LIN {X 0,Y 298.384,Z 335.943,A -85,B 0,C 180,E1 -16518.911,E2 -16518.911} C_VEL
LIN {X 0,Y 298.442,Z 335.935,A -85,B 0,C 180,E1 -16523.191,E2 -16523.191} C_VEL
LIN {X 0,Y 298.393,Z 335.94,A -85,B 0,C 180,E1 -16527.199,E2 -16527.199} C_VEL
LIN {X 0,Y 298.428,Z 335.937,A -85,B 0,C 180,E1 -16530.613,E2 -16530.613} C_VEL
LIN {X 0,Y 298.478,Z 335.928,A -85,B 0,C 180,E1 -16533.473,E2 -16533.473} C_VEL
LIN {X 0,Y 298.429,Z 335.938,A -85,B 0,C 180,E1 -16536.696,E2 -16536.696} C_VEL
LIN {X 0,Y 298.533,Z 335.925,A -85,B 0,C 180,E1 -16540.756,E2 -16540.756} C_VEL
LIN {X 0,Y 298.586,Z 335.915,A -85,B 0,C 180,E1 -16544.994,E2 -16544.994} C_VEL
LIN {X 0,Y 298.586,Z 335.915,A -85,B 0,C 180,E1 -16549.146,E2 -16549.146} C_VEL
LIN {X 0,Y 298.753,Z 335.894,A -85,B 0,C 180,E1 -16551.885,E2 -16551.885} C_VEL
LIN {X 0,Y 298.654,Z 335.909,A -85,B 0,C 180,E1 -16554.598,E2 -16554.598} C_VEL
LIN {X 0,Y 298.916,Z 335.876,A -85,B 0,C 180,E1 -16558.652,E2 -16558.652} C_VEL
LIN {X 0,Y 298.918,Z 335.872,A -85,B 0,C 180,E1 -16561.347,E2 -16561.347} C_VEL
LIN {X 0,Y 298.785,Z 335.89,A -85,B 0,C 180,E1 -16562.896,E2 -16562.896} C_VEL
LIN {X 0,Y 297.957,Z 335.996,A -85,B 0,C 180,E1 -16564.02,E2 -16564.02} C_VEL
LIN {X 0,Y 295.074,Z 336.353,A -85,B 0,C 180,E1 -16565.854,E2 -16565.854} C_VEL
LIN {X 0,Y 292.741,Z 336.645,A -85,B 0,C 180,E1 -16567.341,E2 -16567.341} C_VEL
LIN {X 0,Y 291.768,Z 336.766,A -85,B 0,C 180,E1 -16568.492,E2 -16568.492} C_VEL
LIN {X 0,Y 291.696,Z 336.772,A -85,B 0,C 180,E1 -16568.881,E2 -16568.881} C_VEL
LIN {X 0,Y 291.515,Z 336.798,A -85,B 0,C 180,E1 -16573.95,E2 -16573.95} C_VEL
LIN {X 0,Y 291.48,Z 336.799,A -85,B 0,C 180,E1 -16576.818,E2 -16576.818} C_VEL
LIN {X 0,Y 291.443,Z 336.806,A -85,B 0,C 180,E1 -16579.875,E2 -16579.875} C_VEL
LIN {X 0,Y 291.393,Z 336.813,A -85,B 0,C 180,E1 -16584.206,E2 -16584.206} C_VEL
LIN {X 0,Y 291.415,Z 336.807,A -85,B 0,C 180,E1 -16587.272,E2 -16587.272} C_VEL
LIN {X 0,Y 291.332,Z 336.819,A -85,B 0,C 180,E1 -16590.437,E2 -16590.437} C_VEL
LIN {X 0,Y 291.339,Z 336.821,A -85,B 0,C 180,E1 -16593.699,E2 -16593.699} C_VEL
LIN {X 0,Y 291.431,Z 336.915,A -85,B 0,C 180,E1 -16596.753,E2 -16596.753} C_VEL
LIN {X 0,Y 292.734,Z 343.937,A -85,B 0,C 180,E1 -16600.407,E2 -16600.407} C_VEL
LIN {X 0,Y 294.252,Z 351.677,A -85,B 0,C 180,E1 -16604.234,E2 -16604.234} C_VEL
LIN {X 0,Y 296.055,Z 360.385,A -85,B 0,C 180,E1 -16608.344,E2 -16608.344} C_VEL
LIN {X 0,Y 296.139,Z 362.771,A -85,B 0,C 180,E1 -16609.413,E2 -16609.413} C_VEL
LIN {X 0,Y 294.612,Z 372.008,A -85,B 0,C 180,E1 -16613.391,E2 -16613.391} C_VEL
LIN {X 0,Y 293.002,Z 383.21,A -85,B 0,C 180,E1 -16618.152,E2 -16618.152} C_VEL
LIN {X 0,Y 291.754,Z 394.182,A -85,B 0,C 180,E1 -16622.764,E2 -16622.764} C_VEL
LIN {X 0,Y 291.663,Z 395.459,A -85,B 0,C 180,E1 -16623.189,E2 -16623.189} C_VEL
LIN {X 0,Y 293.313,Z 416.036,A -85,B 0,C 180,E1 -16624.452,E2 -16624.452} C_VEL
LIN {X 0,Y 294.42,Z 430.699,A -85,B 0,C 180,E1 -16625.619,E2 -16625.619} C_VEL
LIN {X 0,Y 295.568,Z 445.292,A -85,B 0,C 180,E1 -16627.087,E2 -16627.087} C_VEL
LIN {X 0,Y 296.15,Z 455.041,A -85,B 0,C 180,E1 -16628.237,E2 -16628.237} C_VEL
LIN {X 0,Y 294.693,Z 467.515,A -85,B 0,C 180,E1 -16629.953,E2 -16629.953} C_VEL
LIN {X 0,Y 293.284,Z 478.836,A -85,B 0,C 180,E1 -16631.851,E2 -16631.851} C_VEL
LIN {X 0,Y 292.138,Z 489.112,A -85,B 0,C 180,E1 -16633.941,E2 -16633.941} C_VEL
LIN {X 0,Y 291.317,Z 497.647,A -85,B 0,C 180,E1 -16636.041,E2 -16636.041} C_VEL
LIN {X 0,Y 290.887,Z 505.868,A -85,B 0,C 180,E1 -16638.504,E2 -16638.504} C_VEL
LIN {X 0,Y 290.817,Z 512.39,A -85,B 0,C 180,E1 -16640.964,E2 -16640.964} C_VEL
LIN {X 0,Y 291.047,Z 516.816,A -85,B 0,C 180,E1 -16643.067,E2 -16643.067} C_VEL
LIN {X 0,Y 291.187,Z 519.192,A -85,B 0,C 180,E1 -16644.461,E2 -16644.461} C_VEL
LIN {X 0,Y 291.509,Z 522.595,A -85,B 0,C 180,E1 -16647.238,E2 -16647.238} C_VEL
LIN {X 0,Y 291.68,Z 523.685,A -85,B 0,C 180,E1 -16648.621,E2 -16648.621} C_VEL
LIN {X 0,Y 291.849,Z 524.383,A -85,B 0,C 180,E1 -16650.001,E2 -16650.001} C_VEL
LIN {X 0,Y 291.523,Z 524.606,A -85,B 0,C 180,E1 -16651.383,E2 -16651.383} C_VEL
LIN {X 0,Y 290.918,Z 523.938,A -85,B 0,C 180,E1 -16654.157,E2 -16654.157} C_VEL
LIN {X 0,Y 290.727,Z 523.064,A -85,B 0,C 180,E1 -16655.55,E2 -16655.55} C_VEL
LIN {X 0,Y 290.281,Z 520.217,A -85,B 0,C 180,E1 -16658.354,E2 -16658.354} C_VEL
LIN {X 0,Y 290.24,Z 515.983,A -85,B 0,C 180,E1 -16661.171,E2 -16661.171} C_VEL
LIN {X 0,Y 290.843,Z 510.353,A -85,B 0,C 180,E1 -16663.985,E2 -16663.985} C_VEL
LIN {X 0,Y 292.262,Z 503.283,A -85,B 0,C 180,E1 -16666.773,E2 -16666.773} C_VEL
LIN {X 0,Y 294.433,Z 494.668,A -85,B 0,C 180,E1 -16669.523,E2 -16669.523} C_VEL
LIN {X 0,Y 297.551,Z 484.315,A -85,B 0,C 180,E1 -16672.206,E2 -16672.206} C_VEL
LIN {X 0,Y 300.623,Z 474.827,A -85,B 0,C 180,E1 -16674.253,E2 -16674.253} C_VEL
LIN {X 0,Y 303.764,Z 464.971,A -85,B 0,C 180,E1 -16676.079,E2 -16676.079} C_VEL
LIN {X 0,Y 307.037,Z 451.397,A -85,B 0,C 180,E1 -16678.358,E2 -16678.358} C_VEL
LIN {X 0,Y 309.072,Z 440.707,A -85,B 0,C 180,E1 -16680.018,E2 -16680.018} C_VEL
LIN {X 0,Y 310.207,Z 429.791,A -85,B 0,C 180,E1 -16681.737,E2 -16681.737} C_VEL
LIN {X 0,Y 310.622,Z 419.575,A -85,B 0,C 180,E1 -16683.437,E2 -16683.437} C_VEL
LIN {X 0,Y 310.565,Z 410.326,A -85,B 0,C 180,E1 -16685.096,E2 -16685.096} C_VEL
LIN {X 0,Y 310.075,Z 400.116,A -85,B 0,C 180,E1 -16687.159,E2 -16687.159} C_VEL
LIN {X 0,Y 309.74,Z 393.575,A -85,B 0,C 180,E1 -16688.649,E2 -16688.649} C_VEL
LIN {X 0,Y 309.457,Z 385.456,A -85,B 0,C 180,E1 -16690.737,E2 -16690.737} C_VEL
LIN {X 0,Y 309.469,Z 380.582,A -85,B 0,C 180,E1 -16692.221,E2 -16692.221} C_VEL
LIN {X 0,Y 309.456,Z 378.608,A -85,B 0,C 180,E1 -16692.948,E2 -16692.948} C_VEL
LIN {X 0,Y 309.152,Z 375.079,A -85,B 0,C 180,E1 -16695.193,E2 -16695.193} C_VEL
LIN {X 0,Y 309.337,Z 373.381,A -85,B 0,C 180,E1 -16697.032,E2 -16697.032} C_VEL
LIN {X 0,Y 310.764,Z 372.281,A -85,B 0,C 180,E1 -16700.258,E2 -16700.258} C_VEL
LIN {X 0,Y 312.772,Z 372.924,A -85,B 0,C 180,E1 -16702.65,E2 -16702.65} C_VEL
LIN {X 0,Y 314.831,Z 374.395,A -85,B 0,C 180,E1 -16704.522,E2 -16704.522} C_VEL
LIN {X 0,Y 317.095,Z 376.765,A -85,B 0,C 180,E1 -16706.352,E2 -16706.352} C_VEL
LIN {X 0,Y 318.444,Z 379.308,A -85,B 0,C 180,E1 -16707.599,E2 -16707.599} C_VEL
LIN {X 0,Y 319.816,Z 385.394,A -85,B 0,C 180,E1 -16709.641,E2 -16709.641} C_VEL
LIN {X 0,Y 320.499,Z 391.158,A -85,B 0,C 180,E1 -16711.3,E2 -16711.3} C_VEL
LIN {X 0,Y 316.891,Z 401.154,A -85,B 0,C 180,E1 -16712.958,E2 -16712.958} C_VEL
LIN {X 0,Y 312.724,Z 411.585,A -85,B 0,C 180,E1 -16715.079,E2 -16715.079} C_VEL
LIN {X 0,Y 308.879,Z 420.286,A -85,B 0,C 180,E1 -16717.244,E2 -16717.244} C_VEL
LIN {X 0,Y 305.859,Z 426.538,A -85,B 0,C 180,E1 -16719.136,E2 -16719.136} C_VEL
LIN {X 0,Y 302.504,Z 433.284,A -85,B 0,C 180,E1 -16721.721,E2 -16721.721} C_VEL
LIN {X 0,Y 299.864,Z 438.042,A -85,B 0,C 180,E1 -16724.09,E2 -16724.09} C_VEL
LIN {X 0,Y 297.743,Z 441.439,A -85,B 0,C 180,E1 -16726.347,E2 -16726.347} C_VEL
LIN {X 0,Y 295.668,Z 444.227,A -85,B 0,C 180,E1 -16729.038,E2 -16729.038} C_VEL
LIN {X 0,Y 294.017,Z 445.702,A -85,B 0,C 180,E1 -16731.755,E2 -16731.755} C_VEL
LIN {X 0,Y 292.837,Z 445.876,A -85,B 0,C 180,E1 -16734.492,E2 -16734.492} C_VEL
LIN {X 0,Y 292.076,Z 444.754,A -85,B 0,C 180,E1 -16737.242,E2 -16737.242} C_VEL
LIN {X 0,Y 291.759,Z 442.304,A -85,B 0,C 180,E1 -16740,E2 -16740} C_VEL
LIN {X 0,Y 291.643,Z 439.625,A -85,B 0,C 180,E1 -16742.072,E2 -16742.072} C_VEL
LIN {X 0,Y 291.566,Z 434.76,A -85,B 0,C 180,E1 -16744.84,E2 -16744.84} C_VEL
LIN {X 0,Y 292.038,Z 430.099,A -85,B 0,C 180,E1 -16746.911,E2 -16746.911} C_VEL
LIN {X 0,Y 292.606,Z 423.431,A -85,B 0,C 180,E1 -16749.331,E2 -16749.331} C_VEL
LIN {X 0,Y 293.372,Z 415.255,A -85,B 0,C 180,E1 -16751.749,E2 -16751.749} C_VEL
LIN {X 0,Y 294.492,Z 405.302,A -85,B 0,C 180,E1 -16754.159,E2 -16754.159} C_VEL
LIN {X 0,Y 295.596,Z 395.056,A -85,B 0,C 180,E1 -16756.223,E2 -16756.223} C_VEL
LIN {X 0,Y 297.097,Z 382.921,A -85,B 0,C 180,E1 -16758.244,E2 -16758.244} C_VEL
LIN {X 0,Y 298.434,Z 370.378,A -85,B 0,C 180,E1 -16759.967,E2 -16759.967} C_VEL
LIN {X 0,Y 298.882,Z 363.575,A -85,B 0,C 180,E1 -16760.784,E2 -16760.784} C_VEL
LIN {X 0,Y 295.194,Z 350.343,A -85,B 0,C 180,E1 -16762.392,E2 -16762.392} C_VEL
LIN {X 0,Y 291.55,Z 337.403,A -85,B 0,C 180,E1 -16763.773,E2 -16763.773} C_VEL
LIN {X 0,Y 291.45,Z 336.845,A -85,B 0,C 180,E1 -16764.017,E2 -16764.017} C_VEL
LIN {X 0,Y 291.431,Z 336.807,A -85,B 0,C 180,E1 -16767.271,E2 -16767.271} C_VEL
LIN {X 0,Y 291.343,Z 336.82,A -85,B 0,C 180,E1 -16770.437,E2 -16770.437} C_VEL
LIN {X 0,Y 291.35,Z 336.816,A -85,B 0,C 180,E1 -16773.698,E2 -16773.698} C_VEL
LIN {X 0,Y 291.381,Z 336.811,A -85,B 0,C 180,E1 -16777.254,E2 -16777.254} C_VEL
LIN {X 0,Y 291.338,Z 336.821,A -85,B 0,C 180,E1 -16780.642,E2 -16780.642} C_VEL
LIN {X 0,Y 291.296,Z 336.826,A -85,B 0,C 180,E1 -16784.402,E2 -16784.402} C_VEL
LIN {X 0,Y 291.361,Z 336.819,A -85,B 0,C 180,E1 -16788.397,E2 -16788.397} C_VEL
LIN {X 0,Y 291.38,Z 336.812,A -85,B 0,C 180,E1 -16791.161,E2 -16791.161} C_VEL
LIN {X 0,Y 291.392,Z 336.812,A -85,B 0,C 180,E1 -16794.629,E2 -16794.629} C_VEL
LIN {X 0,Y 291.377,Z 336.815,A -85,B 0,C 180,E1 -16797.95,E2 -16797.95} C_VEL
LIN {X 0,Y 291.383,Z 336.811,A -85,B 0,C 180,E1 -16801.157,E2 -16801.157} C_VEL
LIN {X 0,Y 291.42,Z 336.811,A -85,B 0,C 180,E1 -16804.271,E2 -16804.271} C_VEL
LIN {X 0,Y 291.38,Z 336.812,A -85,B 0,C 180,E1 -16807.298,E2 -16807.298} C_VEL
LIN {X 0,Y 291.463,Z 336.803,A -85,B 0,C 180,E1 -16810.269,E2 -16810.269} C_VEL
LIN {X 0,Y 291.561,Z 336.79,A -85,B 0,C 180,E1 -16814.623,E2 -16814.623} C_VEL
LIN {X 0,Y 291.542,Z 336.79,A -85,B 0,C 180,E1 -16818.88,E2 -16818.88} C_VEL
LIN {X 0,Y 291.714,Z 336.773,A -85,B 0,C 180,E1 -16821.687,E2 -16821.687} C_VEL
LIN {X 0,Y 291.635,Z 336.78,A -85,B 0,C 180,E1 -16824.467,E2 -16824.467} C_VEL
LIN {X 0,Y 291.893,Z 336.747,A -85,B 0,C 180,E1 -16828.619,E2 -16828.619} C_VEL
LIN {X 0,Y 291.893,Z 336.75,A -85,B 0,C 180,E1 -16831.378,E2 -16831.378} C_VEL
LIN {X 0,Y 291.75,Z 336.765,A -85,B 0,C 180,E1 -16836.916,E2 -16836.916} C_VEL
LIN {X 0,Y 291.632,Z 336.784,A -85,B 0,C 180,E1 -16839.71,E2 -16839.71} C_VEL
LIN {X 0,Y 291.525,Z 336.794,A -85,B 0,C 180,E1 -16843.949,E2 -16843.949} C_VEL
LIN {X 0,Y 291.489,Z 336.798,A -85,B 0,C 180,E1 -16846.816,E2 -16846.816} C_VEL
LIN {X 0,Y 291.452,Z 336.804,A -85,B 0,C 180,E1 -16849.873,E2 -16849.873} C_VEL
LIN {X 0,Y 291.4,Z 336.809,A -85,B 0,C 180,E1 -16854.204,E2 -16854.204} C_VEL
LIN {X 0,Y 291.419,Z 336.811,A -85,B 0,C 180,E1 -16857.27,E2 -16857.27} C_VEL
LIN {X 0,Y 291.334,Z 336.817,A -85,B 0,C 180,E1 -16860.436,E2 -16860.436} C_VEL
LIN {X 0,Y 291.343,Z 336.818,A -85,B 0,C 180,E1 -16863.697,E2 -16863.697} C_VEL
LIN {X 0,Y 291.371,Z 336.817,A -85,B 0,C 180,E1 -16867.252,E2 -16867.252} C_VEL
LIN {X 0,Y 291.33,Z 336.818,A -85,B 0,C 180,E1 -16870.641,E2 -16870.641} C_VEL
LIN {X 0,Y 291.31,Z 336.821,A -85,B 0,C 180,E1 -16874.396,E2 -16874.396} C_VEL
LIN {X 0,Y 291.323,Z 336.819,A -85,B 0,C 180,E1 -16878.403,E2 -16878.403} C_VEL
LIN {X 0,Y 291.349,Z 336.819,A -85,B 0,C 180,E1 -16881.157,E2 -16881.157} C_VEL
LIN {X 0,Y 291.356,Z 336.817,A -85,B 0,C 180,E1 -16884.625,E2 -16884.625} C_VEL
LIN {X 0,Y 291.37,Z 336.812,A -85,B 0,C 180,E1 -16887.95,E2 -16887.95} C_VEL
LIN {X 0,Y 291.378,Z 336.814,A -85,B 0,C 180,E1 -16891.157,E2 -16891.157} C_VEL
LIN {X 0,Y 291.411,Z 336.809,A -85,B 0,C 180,E1 -16894.271,E2 -16894.271} C_VEL
LIN {X 0,Y 291.376,Z 336.813,A -85,B 0,C 180,E1 -16897.299,E2 -16897.299} C_VEL
LIN {X 0,Y 291.451,Z 336.805,A -85,B 0,C 180,E1 -16900.269,E2 -16900.269} C_VEL
LIN {X 0,Y 291.548,Z 336.795,A -85,B 0,C 180,E1 -16904.623,E2 -16904.623} C_VEL
LIN {X 0,Y 291.53,Z 336.795,A -85,B 0,C 180,E1 -16908.88,E2 -16908.88} C_VEL
LIN {X 0,Y 291.703,Z 336.771,A -85,B 0,C 180,E1 -16911.688,E2 -16911.688} C_VEL
LIN {X 0,Y 291.625,Z 336.785,A -85,B 0,C 180,E1 -16914.468,E2 -16914.468} C_VEL
LIN {X 0,Y 291.883,Z 336.752,A -85,B 0,C 180,E1 -16918.62,E2 -16918.62} C_VEL
LIN {X 0,Y 291.884,Z 336.748,A -85,B 0,C 180,E1 -16921.379,E2 -16921.379} C_VEL
LIN {X 0,Y 291.739,Z 336.768,A -85,B 0,C 180,E1 -16926.918,E2 -16926.918} C_VEL
LIN {X 0,Y 291.696,Z 336.772,A -85,B 0,C 180,E1 -16928.881,E2 -16928.881} C_VEL
LIN {X 0,Y 291.026,Z 336.859,A -85,B 0,C 180,E1 -16930.033,E2 -16930.033} C_VEL
LIN {X 0,Y 288.091,Z 337.223,A -85,B 0,C 180,E1 -16931.906,E2 -16931.906} C_VEL
LIN {X 0,Y 285.6,Z 337.534,A -85,B 0,C 180,E1 -16933.427,E2 -16933.427} C_VEL
LIN {X 0,Y 284.543,Z 337.666,A -85,B 0,C 180,E1 -16934.608,E2 -16934.608} C_VEL
LIN {X 0,Y 284.464,Z 337.673,A -85,B 0,C 180,E1 -16935.008,E2 -16935.008} C_VEL
LIN {X 0,Y 284.396,Z 337.681,A -85,B 0,C 180,E1 -16938.739,E2 -16938.739} C_VEL
LIN {X 0,Y 284.359,Z 337.687,A -85,B 0,C 180,E1 -16943.293,E2 -16943.293} C_VEL
LIN {X 0,Y 284.39,Z 337.682,A -85,B 0,C 180,E1 -16947.174,E2 -16947.174} C_VEL
LIN {X 0,Y 284.291,Z 337.695,A -85,B 0,C 180,E1 -16951.275,E2 -16951.275} C_VEL
LIN {X 0,Y 284.356,Z 337.69,A -85,B 0,C 180,E1 -16955.355,E2 -16955.355} C_VEL
LIN {X 0,Y 284.414,Z 337.85,A -85,B 0,C 180,E1 -16956.484,E2 -16956.484} C_VEL
LIN {X 0,Y 285.934,Z 346.081,A -85,B 0,C 180,E1 -16960.841,E2 -16960.841} C_VEL
LIN {X 0,Y 287.642,Z 354.606,A -85,B 0,C 180,E1 -16965.118,E2 -16965.118} C_VEL
LIN {X 0,Y 289.075,Z 361.67,A -85,B 0,C 180,E1 -16968.512,E2 -16968.512} C_VEL
LIN {X 0,Y 288.92,Z 364.669,A -85,B 0,C 180,E1 -16969.865,E2 -16969.865} C_VEL
LIN {X 0,Y 287.32,Z 373.641,A -85,B 0,C 180,E1 -16973.823,E2 -16973.823} C_VEL
LIN {X 0,Y 285.916,Z 383.442,A -85,B 0,C 180,E1 -16978.099,E2 -16978.099} C_VEL
LIN {X 0,Y 284.641,Z 394.497,A -85,B 0,C 180,E1 -16982.794,E2 -16982.794} C_VEL
LIN {X 0,Y 285.142,Z 401.706,A -85,B 0,C 180,E1 -16983.236,E2 -16983.236} C_VEL
LIN {X 0,Y 286.343,Z 416.546,A -85,B 0,C 180,E1 -16984.208,E2 -16984.208} C_VEL
LIN {X 0,Y 287.461,Z 432.159,A -85,B 0,C 180,E1 -16985.539,E2 -16985.539} C_VEL
LIN {X 0,Y 288.566,Z 446.524,A -85,B 0,C 180,E1 -16987.067,E2 -16987.067} C_VEL
LIN {X 0,Y 288.999,Z 456.415,A -85,B 0,C 180,E1 -16988.308,E2 -16988.308} C_VEL
LIN {X 0,Y 287.363,Z 469.079,A -85,B 0,C 180,E1 -16990.165,E2 -16990.165} C_VEL
LIN {X 0,Y 286.009,Z 479.977,A -85,B 0,C 180,E1 -16992.113,E2 -16992.113} C_VEL
LIN {X 0,Y 284.908,Z 489.858,A -85,B 0,C 180,E1 -16994.257,E2 -16994.257} C_VEL
LIN {X 0,Y 284.185,Z 498.091,A -85,B 0,C 180,E1 -16996.413,E2 -16996.413} C_VEL
LIN {X 0,Y 283.861,Z 504.96,A -85,B 0,C 180,E1 -16998.577,E2 -16998.577} C_VEL
LIN {X 0,Y 283.818,Z 510.593,A -85,B 0,C 180,E1 -17000.739,E2 -17000.739} C_VEL
LIN {X 0,Y 284.019,Z 515.128,A -85,B 0,C 180,E1 -17002.894,E2 -17002.894} C_VEL
LIN {X 0,Y 284.245,Z 518.631,A -85,B 0,C 180,E1 -17005.037,E2 -17005.037} C_VEL
LIN {X 0,Y 284.512,Z 521.176,A -85,B 0,C 180,E1 -17007.17,E2 -17007.17} C_VEL
LIN {X 0,Y 284.695,Z 522.34,A -85,B 0,C 180,E1 -17008.587,E2 -17008.587} C_VEL
LIN {X 0,Y 284.862,Z 523.099,A -85,B 0,C 180,E1 -17010.001,E2 -17010.001} C_VEL
LIN {X 0,Y 284.501,Z 523.377,A -85,B 0,C 180,E1 -17011.417,E2 -17011.417} C_VEL
LIN {X 0,Y 283.867,Z 522.826,A -85,B 0,C 180,E1 -17014.261,E2 -17014.261} C_VEL
LIN {X 0,Y 283.664,Z 522.015,A -85,B 0,C 180,E1 -17015.689,E2 -17015.689} C_VEL
LIN {X 0,Y 283.179,Z 519.302,A -85,B 0,C 180,E1 -17018.565,E2 -17018.565} C_VEL
LIN {X 0,Y 283.18,Z 515.227,A -85,B 0,C 180,E1 -17021.453,E2 -17021.453} C_VEL
LIN {X 0,Y 283.878,Z 509.787,A -85,B 0,C 180,E1 -17024.335,E2 -17024.335} C_VEL
LIN {X 0,Y 285.411,Z 502.934,A -85,B 0,C 180,E1 -17027.188,E2 -17027.188} C_VEL
LIN {X 0,Y 287.698,Z 494.586,A -85,B 0,C 180,E1 -17030,E2 -17030} C_VEL
LIN {X 0,Y 290.995,Z 484.598,A -85,B 0,C 180,E1 -17032.733,E2 -17032.733} C_VEL
LIN {X 0,Y 294.157,Z 475.6,A -85,B 0,C 180,E1 -17034.784,E2 -17034.784} C_VEL
LIN {X 0,Y 297.475,Z 466.005,A -85,B 0,C 180,E1 -17036.673,E2 -17036.673} C_VEL
LIN {X 0,Y 301.507,Z 451.11,A -85,B 0,C 180,E1 -17039.309,E2 -17039.309} C_VEL
LIN {X 0,Y 303.718,Z 440.158,A -85,B 0,C 180,E1 -17041.11,E2 -17041.11} C_VEL
LIN {X 0,Y 305.168,Z 427.686,A -85,B 0,C 180,E1 -17043.237,E2 -17043.237} C_VEL
LIN {X 0,Y 305.763,Z 415.971,A -85,B 0,C 180,E1 -17045.396,E2 -17045.396} C_VEL
LIN {X 0,Y 305.801,Z 406.067,A -85,B 0,C 180,E1 -17047.462,E2 -17047.462} C_VEL
LIN {X 0,Y 305.758,Z 398.289,A -85,B 0,C 180,E1 -17049.308,E2 -17049.308} C_VEL
LIN {X 0,Y 305.929,Z 390.966,A -85,B 0,C 180,E1 -17051.249,E2 -17051.249} C_VEL
LIN {X 0,Y 306.187,Z 386.252,A -85,B 0,C 180,E1 -17052.735,E2 -17052.735} C_VEL
LIN {X 0,Y 306.259,Z 384.286,A -85,B 0,C 180,E1 -17053.508,E2 -17053.508} C_VEL
LIN {X 0,Y 306.166,Z 381.437,A -85,B 0,C 180,E1 -17055.367,E2 -17055.367} C_VEL
LIN {X 0,Y 306.376,Z 379.73,A -85,B 0,C 180,E1 -17057.228,E2 -17057.228} C_VEL
LIN {X 0,Y 307.597,Z 378.679,A -85,B 0,C 180,E1 -17060.227,E2 -17060.227} C_VEL
LIN {X 0,Y 309.46,Z 379.193,A -85,B 0,C 180,E1 -17062.644,E2 -17062.644} C_VEL
LIN {X 0,Y 311.184,Z 380.466,A -85,B 0,C 180,E1 -17064.396,E2 -17064.396} C_VEL
LIN {X 0,Y 313.1,Z 382.536,A -85,B 0,C 180,E1 -17066.154,E2 -17066.154} C_VEL
LIN {X 0,Y 313.799,Z 383.681,A -85,B 0,C 180,E1 -17066.841,E2 -17066.841} C_VEL
LIN {X 0,Y 314.759,Z 388.181,A -85,B 0,C 180,E1 -17068.564,E2 -17068.564} C_VEL
LIN {X 0,Y 315.385,Z 393.682,A -85,B 0,C 180,E1 -17070.352,E2 -17070.352} C_VEL
LIN {X 0,Y 315.358,Z 394.716,A -85,B 0,C 180,E1 -17070.641,E2 -17070.641} C_VEL
LIN {X 0,Y 311.502,Z 404.333,A -85,B 0,C 180,E1 -17072.318,E2 -17072.318} C_VEL
LIN {X 0,Y 306.887,Z 414.87,A -85,B 0,C 180,E1 -17074.571,E2 -17074.571} C_VEL
LIN {X 0,Y 302.852,Z 423.182,A -85,B 0,C 180,E1 -17076.765,E2 -17076.765} C_VEL
LIN {X 0,Y 299.687,Z 429.143,A -85,B 0,C 180,E1 -17078.685,E2 -17078.685} C_VEL
LIN {X 0,Y 296.129,Z 435.545,A -85,B 0,C 180,E1 -17081.314,E2 -17081.314} C_VEL
LIN {X 0,Y 293.115,Z 440.386,A -85,B 0,C 180,E1 -17083.945,E2 -17083.945} C_VEL
LIN {X 0,Y 291.096,Z 443.279,A -85,B 0,C 180,E1 -17086.029,E2 -17086.029} C_VEL
LIN {X 0,Y 288.881,Z 445.824,A -85,B 0,C 180,E1 -17088.777,E2 -17088.777} C_VEL
LIN {X 0,Y 287.127,Z 447.093,A -85,B 0,C 180,E1 -17091.555,E2 -17091.555} C_VEL
LIN {X 0,Y 285.87,Z 447.083,A -85,B 0,C 180,E1 -17094.357,E2 -17094.357} C_VEL
LIN {X 0,Y 285.062,Z 445.784,A -85,B 0,C 180,E1 -17097.174,E2 -17097.174} C_VEL
LIN {X 0,Y 284.735,Z 443.163,A -85,B 0,C 180,E1 -17100,E2 -17100} C_VEL
LIN {X 0,Y 284.581,Z 440.331,A -85,B 0,C 180,E1 -17102.123,E2 -17102.123} C_VEL
LIN {X 0,Y 284.355,Z 436.732,A -85,B 0,C 180,E1 -17104.253,E2 -17104.253} C_VEL
LIN {X 0,Y 285.018,Z 430.476,A -85,B 0,C 180,E1 -17107.082,E2 -17107.082} C_VEL
LIN {X 0,Y 285.686,Z 422.524,A -85,B 0,C 180,E1 -17109.916,E2 -17109.916} C_VEL
LIN {X 0,Y 286.56,Z 413.933,A -85,B 0,C 180,E1 -17112.392,E2 -17112.392} C_VEL
LIN {X 0,Y 287.566,Z 405.099,A -85,B 0,C 180,E1 -17114.508,E2 -17114.508} C_VEL
LIN {X 0,Y 288.736,Z 394.623,A -85,B 0,C 180,E1 -17116.619,E2 -17116.619} C_VEL
LIN {X 0,Y 290.253,Z 382.41,A -85,B 0,C 180,E1 -17118.644,E2 -17118.644} C_VEL
LIN {X 0,Y 291.665,Z 369.239,A -85,B 0,C 180,E1 -17120.451,E2 -17120.451} C_VEL
LIN {X 0,Y 291.914,Z 364.846,A -85,B 0,C 180,E1 -17120.986,E2 -17120.986} C_VEL
LIN {X 0,Y 288.439,Z 352.306,A -85,B 0,C 180,E1 -17122.56,E2 -17122.56} C_VEL
LIN {X 0,Y 284.538,Z 338.361,A -85,B 0,C 180,E1 -17124.085,E2 -17124.085} C_VEL
LIN {X 0,Y 284.401,Z 337.718,A -85,B 0,C 180,E1 -17124.367,E2 -17124.367} C_VEL
LIN {X 0,Y 284.34,Z 337.691,A -85,B 0,C 180,E1 -17128.01,E2 -17128.01} C_VEL
LIN {X 0,Y 284.301,Z 337.695,A -85,B 0,C 180,E1 -17131.274,E2 -17131.274} C_VEL
LIN {X 0,Y 284.346,Z 337.688,A -85,B 0,C 180,E1 -17135.348,E2 -17135.348} C_VEL
LIN {X 0,Y 284.318,Z 337.693,A -85,B 0,C 180,E1 -17138.169,E2 -17138.169} C_VEL
LIN {X 0,Y 284.275,Z 337.699,A -85,B 0,C 180,E1 -17142.124,E2 -17142.124} C_VEL
LIN {X 0,Y 284.278,Z 337.698,A -85,B 0,C 180,E1 -17146.192,E2 -17146.192} C_VEL
LIN {X 0,Y 284.357,Z 337.689,A -85,B 0,C 180,E1 -17150.013,E2 -17150.013} C_VEL
LIN {X 0,Y 284.36,Z 337.686,A -85,B 0,C 180,E1 -17153.617,E2 -17153.617} C_VEL
LIN {X 0,Y 284.313,Z 337.692,A -85,B 0,C 180,E1 -17157.189,E2 -17157.189} C_VEL
LIN {X 0,Y 284.361,Z 337.689,A -85,B 0,C 180,E1 -17160.375,E2 -17160.375} C_VEL
LIN {X 0,Y 284.381,Z 337.684,A -85,B 0,C 180,E1 -17163.586,E2 -17163.586} C_VEL
LIN {X 0,Y 284.339,Z 337.69,A -85,B 0,C 180,E1 -17166.703,E2 -17166.703} C_VEL
LIN {X 0,Y 284.409,Z 337.679,A -85,B 0,C 180,E1 -17171.261,E2 -17171.261} C_VEL
LIN {X 0,Y 284.498,Z 337.67,A -85,B 0,C 180,E1 -17174.458,E2 -17174.458} C_VEL
LIN {X 0,Y 284.494,Z 337.669,A -85,B 0,C 180,E1 -17178.6,E2 -17178.6} C_VEL
LIN {X 0,Y 284.665,Z 337.65,A -85,B 0,C 180,E1 -17181.48,E2 -17181.48} C_VEL
LIN {X 0,Y 284.606,Z 337.657,A -85,B 0,C 180,E1 -17184.33,E2 -17184.33} C_VEL
LIN {X 0,Y 284.859,Z 337.623,A -85,B 0,C 180,E1 -17188.585,E2 -17188.585} C_VEL
LIN {X 0,Y 284.859,Z 337.626,A -85,B 0,C 180,E1 -17191.412,E2 -17191.412} C_VEL
LIN {X 0,Y 284.702,Z 337.643,A -85,B 0,C 180,E1 -17197.089,E2 -17197.089} C_VEL
LIN {X 0,Y 284.57,Z 337.662,A -85,B 0,C 180,E1 -17199.954,E2 -17199.954} C_VEL
LIN {X 0,Y 284.484,Z 337.67,A -85,B 0,C 180,E1 -17204.301,E2 -17204.301} C_VEL
LIN {X 0,Y 284.427,Z 337.68,A -85,B 0,C 180,E1 -17207.247,E2 -17207.247} C_VEL
LIN {X 0,Y 284.38,Z 337.684,A -85,B 0,C 180,E1 -17210.241,E2 -17210.241} C_VEL
LIN {X 0,Y 284.37,Z 337.685,A -85,B 0,C 180,E1 -17213.874,E2 -17213.874} C_VEL
LIN {X 0,Y 284.394,Z 337.685,A -85,B 0,C 180,E1 -17217.171,E2 -17217.171} C_VEL
LIN {X 0,Y 284.293,Z 337.698,A -85,B 0,C 180,E1 -17221.273,E2 -17221.273} C_VEL
LIN {X 0,Y 284.339,Z 337.693,A -85,B 0,C 180,E1 -17225.346,E2 -17225.346} C_VEL
LIN {X 0,Y 284.306,Z 337.693,A -85,B 0,C 180,E1 -17228.168,E2 -17228.168} C_VEL
LIN {X 0,Y 284.267,Z 337.697,A -85,B 0,C 180,E1 -17232.123,E2 -17232.123} C_VEL
LIN {X 0,Y 284.265,Z 337.698,A -85,B 0,C 180,E1 -17236.19,E2 -17236.19} C_VEL
LIN {X 0,Y 284.302,Z 337.692,A -85,B 0,C 180,E1 -17240.022,E2 -17240.022} C_VEL
LIN {X 0,Y 284.328,Z 337.691,A -85,B 0,C 180,E1 -17243.613,E2 -17243.613} C_VEL
LIN {X 0,Y 284.304,Z 337.694,A -85,B 0,C 180,E1 -17247.188,E2 -17247.188} C_VEL
LIN {X 0,Y 284.354,Z 337.688,A -85,B 0,C 180,E1 -17250.375,E2 -17250.375} C_VEL
LIN {X 0,Y 284.372,Z 337.685,A -85,B 0,C 180,E1 -17253.586,E2 -17253.586} C_VEL
LIN {X 0,Y 284.361,Z 337.69,A -85,B 0,C 180,E1 -17256.706,E2 -17256.706} C_VEL
LIN {X 0,Y 284.397,Z 337.682,A -85,B 0,C 180,E1 -17261.261,E2 -17261.261} C_VEL
LIN {X 0,Y 284.485,Z 337.674,A -85,B 0,C 180,E1 -17264.458,E2 -17264.458} C_VEL
LIN {X 0,Y 284.481,Z 337.676,A -85,B 0,C 180,E1 -17268.601,E2 -17268.601} C_VEL
LIN {X 0,Y 284.653,Z 337.649,A -85,B 0,C 180,E1 -17271.481,E2 -17271.481} C_VEL
LIN {X 0,Y 284.595,Z 337.659,A -85,B 0,C 180,E1 -17274.331,E2 -17274.331} C_VEL
LIN {X 0,Y 284.849,Z 337.629,A -85,B 0,C 180,E1 -17278.586,E2 -17278.586} C_VEL
LIN {X 0,Y 284.85,Z 337.624,A -85,B 0,C 180,E1 -17281.413,E2 -17281.413} C_VEL
LIN {X 0,Y 284.691,Z 337.645,A -85,B 0,C 180,E1 -17287.09,E2 -17287.09} C_VEL
LIN {X 0,Y 284.559,Z 337.663,A -85,B 0,C 180,E1 -17289.955,E2 -17289.955} C_VEL
LIN {X 0,Y 284.475,Z 337.676,A -85,B 0,C 180,E1 -17294.303,E2 -17294.303} C_VEL
LIN {X 0,Y 284.464,Z 337.673,A -85,B 0,C 180,E1 -17295.008,E2 -17295.008} C_VEL
LIN {X 0,Y 283.805,Z 337.76,A -85,B 0,C 180,E1 -17296.19,E2 -17296.19} C_VEL
LIN {X 0,Y 280.909,Z 338.12,A -85,B 0,C 180,E1 -17298.112,E2 -17298.112} C_VEL
LIN {X 0,Y 278.43,Z 338.426,A -85,B 0,C 180,E1 -17299.674,E2 -17299.674} C_VEL
LIN {X 0,Y 277.354,Z 338.559,A -85,B 0,C 180,E1 -17300.885,E2 -17300.885} C_VEL
LIN {X 0,Y 277.26,Z 338.569,A -85,B 0,C 180,E1 -17301.296,E2 -17301.296} C_VEL
LIN {X 0,Y 277.312,Z 338.568,A -85,B 0,C 180,E1 -17304.171,E2 -17304.171} C_VEL
LIN {X 0,Y 277.319,Z 338.564,A -85,B 0,C 180,E1 -17307.506,E2 -17307.506} C_VEL
LIN {X 0,Y 277.265,Z 338.571,A -85,B 0,C 180,E1 -17310.482,E2 -17310.482} C_VEL
LIN {X 0,Y 277.248,Z 338.577,A -85,B 0,C 180,E1 -17313.895,E2 -17313.895} C_VEL
LIN {X 0,Y 277.35,Z 338.649,A -85,B 0,C 180,E1 -17316.12,E2 -17316.12} C_VEL
LIN {X 0,Y 278.649,Z 345.78,A -85,B 0,C 180,E1 -17320.022,E2 -17320.022} C_VEL
LIN {X 0,Y 280.385,Z 354.574,A -85,B 0,C 180,E1 -17324.574,E2 -17324.574} C_VEL
LIN {X 0,Y 281.994,Z 362.314,A -85,B 0,C 180,E1 -17328.389,E2 -17328.389} C_VEL
LIN {X 0,Y 281.917,Z 364.901,A -85,B 0,C 180,E1 -17329.599,E2 -17329.599} C_VEL
LIN {X 0,Y 280.445,Z 373.075,A -85,B 0,C 180,E1 -17333.314,E2 -17333.314} C_VEL
LIN {X 0,Y 278.834,Z 383.615,A -85,B 0,C 180,E1 -17338.043,E2 -17338.043} C_VEL
LIN {X 0,Y 277.636,Z 393.612,A -85,B 0,C 180,E1 -17342.406,E2 -17342.406} C_VEL
LIN {X 0,Y 279.204,Z 415.24,A -85,B 0,C 180,E1 -17343.836,E2 -17343.836} C_VEL
LIN {X 0,Y 280.277,Z 430.557,A -85,B 0,C 180,E1 -17345.166,E2 -17345.166} C_VEL
LIN {X 0,Y 281.344,Z 445.028,A -85,B 0,C 180,E1 -17346.736,E2 -17346.736} C_VEL
LIN {X 0,Y 282.006,Z 455.247,A -85,B 0,C 180,E1 -17348.05,E2 -17348.05} C_VEL
LIN {X 0,Y 280.476,Z 467.253,A -85,B 0,C 180,E1 -17349.848,E2 -17349.848} C_VEL
LIN {X 0,Y 279.206,Z 477.313,A -85,B 0,C 180,E1 -17351.662,E2 -17351.662} C_VEL
LIN {X 0,Y 278.064,Z 487.463,A -85,B 0,C 180,E1 -17353.859,E2 -17353.859} C_VEL
LIN {X 0,Y 277.244,Z 495.895,A -85,B 0,C 180,E1 -17356.066,E2 -17356.066} C_VEL
LIN {X 0,Y 276.853,Z 504.005,A -85,B 0,C 180,E1 -17358.655,E2 -17358.655} C_VEL
LIN {X 0,Y 276.857,Z 510.422,A -85,B 0,C 180,E1 -17361.241,E2 -17361.241} C_VEL
LIN {X 0,Y 277.09,Z 514.759,A -85,B 0,C 180,E1 -17363.448,E2 -17363.448} C_VEL
LIN {X 0,Y 277.33,Z 518.019,A -85,B 0,C 180,E1 -17365.641,E2 -17365.641} C_VEL
LIN {X 0,Y 277.516,Z 519.675,A -85,B 0,C 180,E1 -17367.098,E2 -17367.098} C_VEL
LIN {X 0,Y 277.729,Z 520.923,A -85,B 0,C 180,E1 -17368.551,E2 -17368.551} C_VEL
LIN {X 0,Y 277.893,Z 521.757,A -85,B 0,C 180,E1 -17370.001,E2 -17370.001} C_VEL
LIN {X 0,Y 277.513,Z 522.1,A -85,B 0,C 180,E1 -17371.452,E2 -17371.452} C_VEL
LIN {X 0,Y 276.818,Z 521.679,A -85,B 0,C 180,E1 -17374.369,E2 -17374.369} C_VEL
LIN {X 0,Y 276.604,Z 520.937,A -85,B 0,C 180,E1 -17375.834,E2 -17375.834} C_VEL
LIN {X 0,Y 276.099,Z 518.363,A -85,B 0,C 180,E1 -17378.786,E2 -17378.786} C_VEL
LIN {X 0,Y 276.129,Z 514.456,A -85,B 0,C 180,E1 -17381.75,E2 -17381.75} C_VEL
LIN {X 0,Y 276.916,Z 509.223,A -85,B 0,C 180,E1 -17384.703,E2 -17384.703} C_VEL
LIN {X 0,Y 278.563,Z 502.624,A -85,B 0,C 180,E1 -17387.624,E2 -17387.624} C_VEL
LIN {X 0,Y 280.996,Z 494.575,A -85,B 0,C 180,E1 -17390.498,E2 -17390.498} C_VEL
LIN {X 0,Y 284.472,Z 484.927,A -85,B 0,C 180,E1 -17393.285,E2 -17393.285} C_VEL
LIN {X 0,Y 287.703,Z 476.484,A -85,B 0,C 180,E1 -17395.334,E2 -17395.334} C_VEL
LIN {X 0,Y 291.231,Z 467.099,A -85,B 0,C 180,E1 -17397.292,E2 -17397.292} C_VEL
LIN {X 0,Y 294.985,Z 454.79,A -85,B 0,C 180,E1 -17399.629,E2 -17399.629} C_VEL
LIN {X 0,Y 297.706,Z 444.068,A -85,B 0,C 180,E1 -17401.503,E2 -17401.503} C_VEL
LIN {X 0,Y 299.414,Z 433.995,A -85,B 0,C 180,E1 -17403.316,E2 -17403.316} C_VEL
LIN {X 0,Y 300.678,Z 422.339,A -85,B 0,C 180,E1 -17405.532,E2 -17405.532} C_VEL
LIN {X 0,Y 301.252,Z 412.463,A -85,B 0,C 180,E1 -17407.646,E2 -17407.646} C_VEL
LIN {X 0,Y 301.681,Z 403.711,A -85,B 0,C 180,E1 -17409.756,E2 -17409.756} C_VEL
LIN {X 0,Y 302.265,Z 395.914,A -85,B 0,C 180,E1 -17411.924,E2 -17411.924} C_VEL
LIN {X 0,Y 302.847,Z 390.814,A -85,B 0,C 180,E1 -17413.651,E2 -17413.651} C_VEL
LIN {X 0,Y 302.902,Z 388.551,A -85,B 0,C 180,E1 -17414.921,E2 -17414.921} C_VEL
LIN {X 0,Y 302.96,Z 387.231,A -85,B 0,C 180,E1 -17415.984,E2 -17415.984} C_VEL
LIN {X 0,Y 303.242,Z 385.792,A -85,B 0,C 180,E1 -17417.873,E2 -17417.873} C_VEL
LIN {X 0,Y 303.959,Z 385.093,A -85,B 0,C 180,E1 -17419.732,E2 -17419.732} C_VEL
LIN {X 0,Y 305.135,Z 385.024,A -85,B 0,C 180,E1 -17421.547,E2 -17421.547} C_VEL
LIN {X 0,Y 306.577,Z 385.824,A -85,B 0,C 180,E1 -17423.414,E2 -17423.414} C_VEL
LIN {X 0,Y 308.252,Z 387.438,A -85,B 0,C 180,E1 -17425.251,E2 -17425.251} C_VEL
LIN {X 0,Y 309.282,Z 388.74,A -85,B 0,C 180,E1 -17426.292,E2 -17426.292} C_VEL
LIN {X 0,Y 309.928,Z 391.527,A -85,B 0,C 180,E1 -17427.579,E2 -17427.579} C_VEL
LIN {X 0,Y 310.367,Z 397.806,A -85,B 0,C 180,E1 -17429.824,E2 -17429.824} C_VEL
LIN {X 0,Y 305.669,Z 408.732,A -85,B 0,C 180,E1 -17431.879,E2 -17431.879} C_VEL
LIN {X 0,Y 301.061,Z 418.182,A -85,B 0,C 180,E1 -17434.043,E2 -17434.043} C_VEL
LIN {X 0,Y 296.264,Z 427.081,A -85,B 0,C 180,E1 -17436.588,E2 -17436.588} C_VEL
LIN {X 0,Y 292.576,Z 433.401,A -85,B 0,C 180,E1 -17438.881,E2 -17438.881} C_VEL
LIN {X 0,Y 288.803,Z 439.286,A -85,B 0,C 180,E1 -17441.636,E2 -17441.636} C_VEL
LIN {X 0,Y 285.824,Z 443.437,A -85,B 0,C 180,E1 -17444.308,E2 -17444.308} C_VEL
LIN {X 0,Y 283.206,Z 446.414,A -85,B 0,C 180,E1 -17447.095,E2 -17447.095} C_VEL
LIN {X 0,Y 281.125,Z 448.105,A -85,B 0,C 180,E1 -17449.922,E2 -17449.922} C_VEL
LIN {X 0,Y 279.506,Z 448.548,A -85,B 0,C 180,E1 -17452.778,E2 -17452.778} C_VEL
LIN {X 0,Y 278.419,Z 447.712,A -85,B 0,C 180,E1 -17455.657,E2 -17455.657} C_VEL
LIN {X 0,Y 277.8,Z 445.573,A -85,B 0,C 180,E1 -17458.551,E2 -17458.551} C_VEL
LIN {X 0,Y 277.637,Z 442.112,A -85,B 0,C 180,E1 -17461.451,E2 -17461.451} C_VEL
LIN {X 0,Y 277.32,Z 437.257,A -85,B 0,C 180,E1 -17464.361,E2 -17464.361} C_VEL
LIN {X 0,Y 277.982,Z 430.809,A -85,B 0,C 180,E1 -17467.263,E2 -17467.263} C_VEL
LIN {X 0,Y 278.604,Z 423.766,A -85,B 0,C 180,E1 -17469.804,E2 -17469.804} C_VEL
LIN {X 0,Y 279.438,Z 415.199,A -85,B 0,C 180,E1 -17472.344,E2 -17472.344} C_VEL
LIN {X 0,Y 280.481,Z 406.405,A -85,B 0,C 180,E1 -17474.512,E2 -17474.512} C_VEL
LIN {X 0,Y 281.639,Z 395.977,A -85,B 0,C 180,E1 -17476.677,E2 -17476.677} C_VEL
LIN {X 0,Y 283.228,Z 383.399,A -85,B 0,C 180,E1 -17478.82,E2 -17478.82} C_VEL
LIN {X 0,Y 284.65,Z 370.782,A -85,B 0,C 180,E1 -17480.6,E2 -17480.6} C_VEL
LIN {X 0,Y 285.001,Z 366.468,A -85,B 0,C 180,E1 -17481.14,E2 -17481.14} C_VEL
LIN {X 0,Y 281.319,Z 353.041,A -85,B 0,C 180,E1 -17482.867,E2 -17482.867} C_VEL
LIN {X 0,Y 277.473,Z 339.217,A -85,B 0,C 180,E1 -17484.415,E2 -17484.415} C_VEL
LIN {X 0,Y 277.359,Z 338.597,A -85,B 0,C 180,E1 -17484.697,E2 -17484.697} C_VEL
LIN {X 0,Y 277.334,Z 338.563,A -85,B 0,C 180,E1 -17487.506,E2 -17487.506} C_VEL
LIN {X 0,Y 277.278,Z 338.573,A -85,B 0,C 180,E1 -17490.481,E2 -17490.481} C_VEL
LIN {X 0,Y 277.253,Z 338.572,A -85,B 0,C 180,E1 -17493.896,E2 -17493.896} C_VEL
LIN {X 0,Y 277.273,Z 338.568,A -85,B 0,C 180,E1 -17497.469,E2 -17497.469} C_VEL
LIN {X 0,Y 277.215,Z 338.577,A -85,B 0,C 180,E1 -17501.236,E2 -17501.236} C_VEL
LIN {X 0,Y 277.212,Z 338.575,A -85,B 0,C 180,E1 -17505.225,E2 -17505.225} C_VEL
LIN {X 0,Y 277.268,Z 338.57,A -85,B 0,C 180,E1 -17509.502,E2 -17509.502} C_VEL
LIN {X 0,Y 277.293,Z 338.568,A -85,B 0,C 180,E1 -17512.533,E2 -17512.533} C_VEL
LIN {X 0,Y 277.26,Z 338.574,A -85,B 0,C 180,E1 -17516.105,E2 -17516.105} C_VEL
LIN {X 0,Y 277.267,Z 338.57,A -85,B 0,C 180,E1 -17519.538,E2 -17519.538} C_VEL
LIN {X 0,Y 277.362,Z 338.557,A -85,B 0,C 180,E1 -17522.863,E2 -17522.863} C_VEL
LIN {X 0,Y 277.303,Z 338.57,A -85,B 0,C 180,E1 -17526.076,E2 -17526.076} C_VEL
LIN {X 0,Y 277.35,Z 338.558,A -85,B 0,C 180,E1 -17530.765,E2 -17530.765} C_VEL
LIN {X 0,Y 277.44,Z 338.549,A -85,B 0,C 180,E1 -17535.325,E2 -17535.325} C_VEL
LIN {X 0,Y 277.512,Z 338.542,A -85,B 0,C 180,E1 -17539.788,E2 -17539.788} C_VEL
LIN {X 0,Y 277.658,Z 338.521,A -85,B 0,C 180,E1 -17542.728,E2 -17542.728} C_VEL
LIN {X 0,Y 277.825,Z 338.499,A -85,B 0,C 180,E1 -17548.549,E2 -17548.549} C_VEL
LIN {X 0,Y 277.825,Z 338.503,A -85,B 0,C 180,E1 -17551.448,E2 -17551.448} C_VEL
LIN {X 0,Y 277.657,Z 338.522,A -85,B 0,C 180,E1 -17557.269,E2 -17557.269} C_VEL
LIN {X 0,Y 277.51,Z 338.54,A -85,B 0,C 180,E1 -17560.21,E2 -17560.21} C_VEL
LIN {X 0,Y 277.437,Z 338.547,A -85,B 0,C 180,E1 -17564.673,E2 -17564.673} C_VEL
LIN {X 0,Y 277.347,Z 338.563,A -85,B 0,C 180,E1 -17569.232,E2 -17569.232} C_VEL
LIN {X 0,Y 277.319,Z 338.562,A -85,B 0,C 180,E1 -17574.169,E2 -17574.169} C_VEL
LIN {X 0,Y 277.323,Z 338.566,A -85,B 0,C 180,E1 -17577.502,E2 -17577.502} C_VEL
LIN {X 0,Y 277.271,Z 338.569,A -85,B 0,C 180,E1 -17580.48,E2 -17580.48} C_VEL
LIN {X 0,Y 277.245,Z 338.573,A -85,B 0,C 180,E1 -17583.894,E2 -17583.894} C_VEL
LIN {X 0,Y 277.263,Z 338.573,A -85,B 0,C 180,E1 -17587.468,E2 -17587.468} C_VEL
LIN {X 0,Y 277.207,Z 338.581,A -85,B 0,C 180,E1 -17591.235,E2 -17591.235} C_VEL
LIN {X 0,Y 277.213,Z 338.58,A -85,B 0,C 180,E1 -17595.222,E2 -17595.222} C_VEL
LIN {X 0,Y 277.219,Z 338.576,A -85,B 0,C 180,E1 -17599.511,E2 -17599.511} C_VEL
LIN {X 0,Y 277.264,Z 338.572,A -85,B 0,C 180,E1 -17602.529,E2 -17602.529} C_VEL
LIN {X 0,Y 277.243,Z 338.573,A -85,B 0,C 180,E1 -17606.103,E2 -17606.103} C_VEL
LIN {X 0,Y 277.256,Z 338.571,A -85,B 0,C 180,E1 -17609.537,E2 -17609.537} C_VEL
LIN {X 0,Y 277.353,Z 338.563,A -85,B 0,C 180,E1 -17612.863,E2 -17612.863} C_VEL
LIN {X 0,Y 277.323,Z 338.562,A -85,B 0,C 180,E1 -17616.078,E2 -17616.078} C_VEL
LIN {X 0,Y 277.338,Z 338.565,A -85,B 0,C 180,E1 -17620.765,E2 -17620.765} C_VEL
LIN {X 0,Y 277.428,Z 338.549,A -85,B 0,C 180,E1 -17625.325,E2 -17625.325} C_VEL
LIN {X 0,Y 277.5,Z 338.541,A -85,B 0,C 180,E1 -17629.788,E2 -17629.788} C_VEL
LIN {X 0,Y 277.647,Z 338.524,A -85,B 0,C 180,E1 -17632.729,E2 -17632.729} C_VEL
LIN {X 0,Y 277.815,Z 338.505,A -85,B 0,C 180,E1 -17638.55,E2 -17638.55} C_VEL
LIN {X 0,Y 277.815,Z 338.5,A -85,B 0,C 180,E1 -17641.449,E2 -17641.449} C_VEL
LIN {X 0,Y 277.646,Z 338.523,A -85,B 0,C 180,E1 -17647.271,E2 -17647.271} C_VEL
LIN {X 0,Y 277.5,Z 338.544,A -85,B 0,C 180,E1 -17650.211,E2 -17650.211} C_VEL
LIN {X 0,Y 277.42,Z 338.551,A -85,B 0,C 180,E1 -17655.006,E2 -17655.006} C_VEL
LIN {X 0,Y 277.337,Z 338.56,A -85,B 0,C 180,E1 -17659.234,E2 -17659.234} C_VEL
LIN {X 0,Y 277.26,Z 338.569,A -85,B 0,C 180,E1 -17661.296,E2 -17661.296} C_VEL
LIN {X 0,Y 276.569,Z 338.659,A -85,B 0,C 180,E1 -17662.509,E2 -17662.509} C_VEL
LIN {X 0,Y 273.695,Z 339.016,A -85,B 0,C 180,E1 -17664.483,E2 -17664.483} C_VEL
LIN {X 0,Y 271.296,Z 339.316,A -85,B 0,C 180,E1 -17666.088,E2 -17666.088} C_VEL
LIN {X 0,Y 270.309,Z 339.436,A -85,B 0,C 180,E1 -17667.332,E2 -17667.332} C_VEL
LIN {X 0,Y 270.25,Z 339.446,A -85,B 0,C 180,E1 -17667.753,E2 -17667.753} C_VEL
LIN {X 0,Y 270.178,Z 339.454,A -85,B 0,C 180,E1 -17671.349,E2 -17671.349} C_VEL
LIN {X 0,Y 270.285,Z 339.562,A -85,B 0,C 180,E1 -17675.851,E2 -17675.851} C_VEL
LIN {X 0,Y 271.746,Z 347.504,A -85,B 0,C 180,E1 -17680.282,E2 -17680.282} C_VEL
LIN {X 0,Y 273.157,Z 354.503,A -85,B 0,C 180,E1 -17684.001,E2 -17684.001} C_VEL
LIN {X 0,Y 274.948,Z 363.086,A -85,B 0,C 180,E1 -17688.351,E2 -17688.351} C_VEL
LIN {X 0,Y 274.567,Z 366.992,A -85,B 0,C 180,E1 -17690.217,E2 -17690.217} C_VEL
LIN {X 0,Y 272.85,Z 376.382,A -85,B 0,C 180,E1 -17694.583,E2 -17694.583} C_VEL
LIN {X 0,Y 271.515,Z 385.553,A -85,B 0,C 180,E1 -17698.825,E2 -17698.825} C_VEL
LIN {X 0,Y 270.643,Z 392.616,A -85,B 0,C 180,E1 -17701.994,E2 -17701.994} C_VEL
LIN {X 0,Y 270.803,Z 396.496,A -85,B 0,C 180,E1 -17702.284,E2 -17702.284} C_VEL
LIN {X 0,Y 271.96,Z 412.159,A -85,B 0,C 180,E1 -17703.322,E2 -17703.322} C_VEL
LIN {X 0,Y 273.009,Z 427.241,A -85,B 0,C 180,E1 -17704.619,E2 -17704.619} C_VEL
LIN {X 0,Y 274.042,Z 441.738,A -85,B 0,C 180,E1 -17706.185,E2 -17706.185} C_VEL
LIN {X 0,Y 274.851,Z 454.438,A -85,B 0,C 180,E1 -17707.844,E2 -17707.844} C_VEL
LIN {X 0,Y 273.945,Z 463.17,A -85,B 0,C 180,E1 -17709.149,E2 -17709.149} C_VEL
LIN {X 0,Y 272.457,Z 474.609,A -85,B 0,C 180,E1 -17711.191,E2 -17711.191} C_VEL
LIN {X 0,Y 271.118,Z 485.477,A -85,B 0,C 180,E1 -17713.561,E2 -17713.561} C_VEL
LIN {X 0,Y 270.216,Z 494.921,A -85,B 0,C 180,E1 -17716.081,E2 -17716.081} C_VEL
LIN {X 0,Y 269.858,Z 502.988,A -85,B 0,C 180,E1 -17718.738,E2 -17718.738} C_VEL
LIN {X 0,Y 269.862,Z 508.564,A -85,B 0,C 180,E1 -17721.012,E2 -17721.012} C_VEL
LIN {X 0,Y 270.076,Z 513.011,A -85,B 0,C 180,E1 -17723.277,E2 -17723.277} C_VEL
LIN {X 0,Y 270.357,Z 516.431,A -85,B 0,C 180,E1 -17725.529,E2 -17725.529} C_VEL
LIN {X 0,Y 270.525,Z 518.153,A -85,B 0,C 180,E1 -17727.023,E2 -17727.023} C_VEL
LIN {X 0,Y 270.756,Z 519.473,A -85,B 0,C 180,E1 -17728.514,E2 -17728.514} C_VEL
LIN {X 0,Y 270.938,Z 520.38,A -85,B 0,C 180,E1 -17730.001,E2 -17730.001} C_VEL
LIN {X 0,Y 270.517,Z 520.781,A -85,B 0,C 180,E1 -17731.49,E2 -17731.49} C_VEL
LIN {X 0,Y 269.775,Z 520.487,A -85,B 0,C 180,E1 -17734.484,E2 -17734.484} C_VEL
LIN {X 0,Y 269.54,Z 519.813,A -85,B 0,C 180,E1 -17735.988,E2 -17735.988} C_VEL
LIN {X 0,Y 269.02,Z 517.391,A -85,B 0,C 180,E1 -17739.019,E2 -17739.019} C_VEL
LIN {X 0,Y 269.091,Z 513.66,A -85,B 0,C 180,E1 -17742.062,E2 -17742.062} C_VEL
LIN {X 0,Y 269.969,Z 508.633,A -85,B 0,C 180,E1 -17745.091,E2 -17745.091} C_VEL
LIN {X 0,Y 271.725,Z 502.272,A -85,B 0,C 180,E1 -17748.083,E2 -17748.083} C_VEL
LIN {X 0,Y 274.321,Z 494.529,A -85,B 0,C 180,E1 -17751.02,E2 -17751.02} C_VEL
LIN {X 0,Y 277.98,Z 485.283,A -85,B 0,C 180,E1 -17753.862,E2 -17753.862} C_VEL
LIN {X 0,Y 281.166,Z 477.524,A -85,B 0,C 180,E1 -17755.862,E2 -17755.862} C_VEL
LIN {X 0,Y 285.022,Z 468.194,A -85,B 0,C 180,E1 -17757.938,E2 -17757.938} C_VEL
LIN {X 0,Y 289.604,Z 454.661,A -85,B 0,C 180,E1 -17760.64,E2 -17760.64} C_VEL
LIN {X 0,Y 292.593,Z 443.792,A -85,B 0,C 180,E1 -17762.665,E2 -17762.665} C_VEL
LIN {X 0,Y 294.79,Z 432.262,A -85,B 0,C 180,E1 -17764.903,E2 -17764.903} C_VEL
LIN {X 0,Y 296.163,Z 421.609,A -85,B 0,C 180,E1 -17767.143,E2 -17767.143} C_VEL
LIN {X 0,Y 297.019,Z 412.858,A -85,B 0,C 180,E1 -17769.23,E2 -17769.23} C_VEL
LIN {X 0,Y 297.653,Z 406.598,A -85,B 0,C 180,E1 -17770.926,E2 -17770.926} C_VEL
LIN {X 0,Y 298.442,Z 401.283,A -85,B 0,C 180,E1 -17772.436,E2 -17772.436} C_VEL
LIN {X 0,Y 299.337,Z 396.087,A -85,B 0,C 180,E1 -17774.281,E2 -17774.281} C_VEL
LIN {X 0,Y 299.45,Z 394.502,A -85,B 0,C 180,E1 -17775.244,E2 -17775.244} C_VEL
LIN {X 0,Y 299.613,Z 392.596,A -85,B 0,C 180,E1 -17777.137,E2 -17777.137} C_VEL
LIN {X 0,Y 300.114,Z 391.536,A -85,B 0,C 180,E1 -17779.028,E2 -17779.028} C_VEL
LIN {X 0,Y 301.072,Z 391.16,A -85,B 0,C 180,E1 -17780.93,E2 -17780.93} C_VEL
LIN {X 0,Y 302.308,Z 391.569,A -85,B 0,C 180,E1 -17782.811,E2 -17782.811} C_VEL
LIN {X 0,Y 303.77,Z 392.799,A -85,B 0,C 180,E1 -17784.662,E2 -17784.662} C_VEL
LIN {X 0,Y 304.949,Z 394.265,A -85,B 0,C 180,E1 -17786.067,E2 -17786.067} C_VEL
LIN {X 0,Y 305.39,Z 397.612,A -85,B 0,C 180,E1 -17787.634,E2 -17787.634} C_VEL
LIN {X 0,Y 305.43,Z 400.699,A -85,B 0,C 180,E1 -17788.829,E2 -17788.829} C_VEL
LIN {X 0,Y 304.997,Z 402.612,A -85,B 0,C 180,E1 -17789.346,E2 -17789.346} C_VEL
LIN {X 0,Y 299.406,Z 413.913,A -85,B 0,C 180,E1 -17791.619,E2 -17791.619} C_VEL
LIN {X 0,Y 294.644,Z 422.674,A -85,B 0,C 180,E1 -17793.815,E2 -17793.815} C_VEL
LIN {X 0,Y 289.625,Z 430.916,A -85,B 0,C 180,E1 -17796.398,E2 -17796.398} C_VEL
LIN {X 0,Y 285.403,Z 437.429,A -85,B 0,C 180,E1 -17799.081,E2 -17799.081} C_VEL
LIN {X 0,Y 281.559,Z 442.667,A -85,B 0,C 180,E1 -17801.919,E2 -17801.919} C_VEL
LIN {X 0,Y 279.261,Z 445.395,A -85,B 0,C 180,E1 -17803.929,E2 -17803.929} C_VEL
LIN {X 0,Y 276.497,Z 448.139,A -85,B 0,C 180,E1 -17806.776,E2 -17806.776} C_VEL
LIN {X 0,Y 274.319,Z 449.609,A -85,B 0,C 180,E1 -17809.669,E2 -17809.669} C_VEL
LIN {X 0,Y 272.581,Z 449.853,A -85,B 0,C 180,E1 -17812.593,E2 -17812.593} C_VEL
LIN {X 0,Y 271.423,Z 448.818,A -85,B 0,C 180,E1 -17815.545,E2 -17815.545} C_VEL
LIN {X 0,Y 270.778,Z 446.471,A -85,B 0,C 180,E1 -17818.513,E2 -17818.513} C_VEL
LIN {X 0,Y 270.59,Z 442.788,A -85,B 0,C 180,E1 -17821.489,E2 -17821.489} C_VEL
LIN {X 0,Y 270.269,Z 437.736,A -85,B 0,C 180,E1 -17824.475,E2 -17824.475} C_VEL
LIN {X 0,Y 270.934,Z 431.099,A -85,B 0,C 180,E1 -17827.453,E2 -17827.453} C_VEL
LIN {X 0,Y 271.599,Z 423.54,A -85,B 0,C 180,E1 -17830.17,E2 -17830.17} C_VEL
LIN {X 0,Y 272.472,Z 415.08,A -85,B 0,C 180,E1 -17832.665,E2 -17832.665} C_VEL
LIN {X 0,Y 273.547,Z 406.042,A -85,B 0,C 180,E1 -17834.888,E2 -17834.888} C_VEL
LIN {X 0,Y 274.789,Z 395.298,A -85,B 0,C 180,E1 -17837.105,E2 -17837.105} C_VEL
LIN {X 0,Y 276.448,Z 382.439,A -85,B 0,C 180,E1 -17839.299,E2 -17839.299} C_VEL
LIN {X 0,Y 277.89,Z 369.48,A -85,B 0,C 180,E1 -17841.125,E2 -17841.125} C_VEL
LIN {X 0,Y 278.009,Z 367.987,A -85,B 0,C 180,E1 -17841.309,E2 -17841.309} C_VEL
LIN {X 0,Y 274.741,Z 355.709,A -85,B 0,C 180,E1 -17842.94,E2 -17842.94} C_VEL
LIN {X 0,Y 270.412,Z 340.084,A -85,B 0,C 180,E1 -17844.757,E2 -17844.757} C_VEL
LIN {X 0,Y 270.296,Z 339.47,A -85,B 0,C 180,E1 -17845.066,E2 -17845.066} C_VEL
LIN {X 0,Y 270.278,Z 339.443,A -85,B 0,C 180,E1 -17847.908,E2 -17847.908} C_VEL
LIN {X 0,Y 270.19,Z 339.452,A -85,B 0,C 180,E1 -17851.348,E2 -17851.348} C_VEL
LIN {X 0,Y 270.208,Z 339.451,A -85,B 0,C 180,E1 -17854.905,E2 -17854.905} C_VEL
LIN {X 0,Y 270.203,Z 339.453,A -85,B 0,C 180,E1 -17858.71,E2 -17858.71} C_VEL
LIN {X 0,Y 270.177,Z 339.456,A -85,B 0,C 180,E1 -17862.558,E2 -17862.558} C_VEL
LIN {X 0,Y 270.186,Z 339.454,A -85,B 0,C 180,E1 -17866.747,E2 -17866.747} C_VEL
LIN {X 0,Y 270.219,Z 339.448,A -85,B 0,C 180,E1 -17869.441,E2 -17869.441} C_VEL
LIN {X 0,Y 270.263,Z 339.442,A -85,B 0,C 180,E1 -17873.721,E2 -17873.721} C_VEL
LIN {X 0,Y 270.21,Z 339.45,A -85,B 0,C 180,E1 -17876.892,E2 -17876.892} C_VEL
LIN {X 0,Y 270.201,Z 339.452,A -85,B 0,C 180,E1 -17880.382,E2 -17880.382} C_VEL
LIN {X 0,Y 270.266,Z 339.443,A -85,B 0,C 180,E1 -17883.763,E2 -17883.763} C_VEL
LIN {X 0,Y 270.216,Z 339.448,A -85,B 0,C 180,E1 -17887.036,E2 -17887.036} C_VEL
LIN {X 0,Y 270.307,Z 339.438,A -85,B 0,C 180,E1 -17890.244,E2 -17890.244} C_VEL
LIN {X 0,Y 270.409,Z 339.424,A -85,B 0,C 180,E1 -17894.934,E2 -17894.934} C_VEL
LIN {X 0,Y 270.447,Z 339.42,A -85,B 0,C 180,E1 -17899.518,E2 -17899.518} C_VEL
LIN {X 0,Y 270.616,Z 339.399,A -85,B 0,C 180,E1 -17902.538,E2 -17902.538} C_VEL
LIN {X 0,Y 270.791,Z 339.376,A -85,B 0,C 180,E1 -17908.511,E2 -17908.511} C_VEL
LIN {X 0,Y 270.791,Z 339.379,A -85,B 0,C 180,E1 -17911.486,E2 -17911.486} C_VEL
LIN {X 0,Y 270.615,Z 339.4,A -85,B 0,C 180,E1 -17917.46,E2 -17917.46} C_VEL
LIN {X 0,Y 270.445,Z 339.42,A -85,B 0,C 180,E1 -17920.479,E2 -17920.479} C_VEL
LIN {X 0,Y 270.405,Z 339.425,A -85,B 0,C 180,E1 -17925.063,E2 -17925.063} C_VEL
LIN {X 0,Y 270.303,Z 339.44,A -85,B 0,C 180,E1 -17929.754,E2 -17929.754} C_VEL
LIN {X 0,Y 270.274,Z 339.44,A -85,B 0,C 180,E1 -17934.584,E2 -17934.584} C_VEL
LIN {X 0,Y 270.269,Z 339.442,A -85,B 0,C 180,E1 -17937.907,E2 -17937.907} C_VEL
LIN {X 0,Y 270.183,Z 339.455,A -85,B 0,C 180,E1 -17941.346,E2 -17941.346} C_VEL
LIN {X 0,Y 270.2,Z 339.452,A -85,B 0,C 180,E1 -17944.904,E2 -17944.904} C_VEL
LIN {X 0,Y 270.195,Z 339.452,A -85,B 0,C 180,E1 -17948.709,E2 -17948.709} C_VEL
LIN {X 0,Y 270.168,Z 339.458,A -85,B 0,C 180,E1 -17953.249,E2 -17953.249} C_VEL
LIN {X 0,Y 270.171,Z 339.454,A -85,B 0,C 180,E1 -17957.441,E2 -17957.441} C_VEL
LIN {X 0,Y 270.203,Z 339.451,A -85,B 0,C 180,E1 -17961.373,E2 -17961.373} C_VEL
LIN {X 0,Y 270.197,Z 339.453,A -85,B 0,C 180,E1 -17965.093,E2 -17965.093} C_VEL
LIN {X 0,Y 270.195,Z 339.453,A -85,B 0,C 180,E1 -17969.129,E2 -17969.129} C_VEL
LIN {X 0,Y 270.259,Z 339.443,A -85,B 0,C 180,E1 -17972.144,E2 -17972.144} C_VEL
LIN {X 0,Y 270.271,Z 339.44,A -85,B 0,C 180,E1 -17975.518,E2 -17975.518} C_VEL
LIN {X 0,Y 270.295,Z 339.44,A -85,B 0,C 180,E1 -17980.243,E2 -17980.243} C_VEL
LIN {X 0,Y 270.396,Z 339.427,A -85,B 0,C 180,E1 -17984.935,E2 -17984.935} C_VEL
LIN {X 0,Y 270.435,Z 339.421,A -85,B 0,C 180,E1 -17989.518,E2 -17989.518} C_VEL
LIN {X 0,Y 270.605,Z 339.402,A -85,B 0,C 180,E1 -17992.538,E2 -17992.538} C_VEL
LIN {X 0,Y 270.78,Z 339.382,A -85,B 0,C 180,E1 -17998.512,E2 -17998.512} C_VEL
LIN {X 0,Y 270.781,Z 339.376,A -85,B 0,C 180,E1 -18001.487,E2 -18001.487} C_VEL
LIN {X 0,Y 270.604,Z 339.4,A -85,B 0,C 180,E1 -18007.461,E2 -18007.461} C_VEL
LIN {X 0,Y 270.435,Z 339.422,A -85,B 0,C 180,E1 -18010.481,E2 -18010.481} C_VEL
LIN {X 0,Y 270.396,Z 339.426,A -85,B 0,C 180,E1 -18015.065,E2 -18015.065} C_VEL
LIN {X 0,Y 270.294,Z 339.439,A -85,B 0,C 180,E1 -18019.756,E2 -18019.756} C_VEL
LIN {X 0,Y 270.267,Z 339.442,A -85,B 0,C 180,E1 -18024.586,E2 -18024.586} C_VEL
LIN {X 0,Y 270.25,Z 339.446,A -85,B 0,C 180,E1 -18027.753,E2 -18027.753} C_VEL
LIN {X 0,Y 269.633,Z 339.53,A -85,B 0,C 180,E1 -18028.996,E2 -18028.996} C_VEL
LIN {X 0,Y 266.772,Z 339.89,A -85,B 0,C 180,E1 -18031.021,E2 -18031.021} C_VEL
LIN {X 0,Y 264.309,Z 340.193,A -85,B 0,C 180,E1 -18032.668,E2 -18032.668} C_VEL
LIN {X 0,Y 263.248,Z 340.321,A -85,B 0,C 180,E1 -18033.945,E2 -18033.945} C_VEL
LIN {X 0,Y 263.162,Z 340.33,A -85,B 0,C 180,E1 -18034.379,E2 -18034.379} C_VEL
LIN {X 0,Y 263.25,Z 340.503,A -85,B 0,C 180,E1 -18035.614,E2 -18035.614} C_VEL
LIN {X 0,Y 264.548,Z 347.471,A -85,B 0,C 180,E1 -18039.612,E2 -18039.612} C_VEL
LIN {X 0,Y 266.139,Z 355.489,A -85,B 0,C 180,E1 -18043.982,E2 -18043.982} C_VEL
LIN {X 0,Y 267.833,Z 363.633,A -85,B 0,C 180,E1 -18048.223,E2 -18048.223} C_VEL
LIN {X 0,Y 267.691,Z 366.395,A -85,B 0,C 180,E1 -18049.585,E2 -18049.585} C_VEL
LIN {X 0,Y 266.121,Z 374.644,A -85,B 0,C 180,E1 -18053.546,E2 -18053.546} C_VEL
LIN {X 0,Y 264.585,Z 384.416,A -85,B 0,C 180,E1 -18058.211,E2 -18058.211} C_VEL
LIN {X 0,Y 263.625,Z 391.795,A -85,B 0,C 180,E1 -18061.612,E2 -18061.612} C_VEL
LIN {X 0,Y 264.039,Z 399.079,A -85,B 0,C 180,E1 -18062.105,E2 -18062.105} C_VEL
LIN {X 0,Y 265.105,Z 414.402,A -85,B 0,C 180,E1 -18063.215,E2 -18063.215} C_VEL
LIN {X 0,Y 266.057,Z 429.088,A -85,B 0,C 180,E1 -18064.591,E2 -18064.591} C_VEL
LIN {X 0,Y 267.125,Z 444.197,A -85,B 0,C 180,E1 -18066.347,E2 -18066.347} C_VEL
LIN {X 0,Y 267.719,Z 456.262,A -85,B 0,C 180,E1 -18068.034,E2 -18068.034} C_VEL
LIN {X 0,Y 266.176,Z 467.697,A -85,B 0,C 180,E1 -18069.927,E2 -18069.927} C_VEL
LIN {X 0,Y 264.938,Z 477.336,A -85,B 0,C 180,E1 -18071.84,E2 -18071.84} C_VEL
LIN {X 0,Y 263.803,Z 487.33,A -85,B 0,C 180,E1 -18074.232,E2 -18074.232} C_VEL
LIN {X 0,Y 263.058,Z 496.348,A -85,B 0,C 180,E1 -18076.876,E2 -18076.876} C_VEL
LIN {X 0,Y 262.839,Z 502.9,A -85,B 0,C 180,E1 -18079.214,E2 -18079.214} C_VEL
LIN {X 0,Y 262.915,Z 508.206,A -85,B 0,C 180,E1 -18081.511,E2 -18081.511} C_VEL
LIN {X 0,Y 263.165,Z 512.554,A -85,B 0,C 180,E1 -18083.869,E2 -18083.869} C_VEL
LIN {X 0,Y 263.379,Z 514.818,A -85,B 0,C 180,E1 -18085.41,E2 -18085.41} C_VEL
LIN {X 0,Y 263.538,Z 516.61,A -85,B 0,C 180,E1 -18086.944,E2 -18086.944} C_VEL
LIN {X 0,Y 263.775,Z 518.003,A -85,B 0,C 180,E1 -18088.475,E2 -18088.475} C_VEL
LIN {X 0,Y 263.972,Z 518.985,A -85,B 0,C 180,E1 -18090.001,E2 -18090.001} C_VEL
LIN {X 0,Y 263.518,Z 519.447,A -85,B 0,C 180,E1 -18091.53,E2 -18091.53} C_VEL
LIN {X 0,Y 262.73,Z 519.29,A -85,B 0,C 180,E1 -18094.604,E2 -18094.604} C_VEL
LIN {X 0,Y 262.182,Z 518,A -85,B 0,C 180,E1 -18097.336,E2 -18097.336} C_VEL
LIN {X 0,Y 261.91,Z 514.813,A -85,B 0,C 180,E1 -18100.828,E2 -18100.828} C_VEL
LIN {X 0,Y 262.413,Z 510.639,A -85,B 0,C 180,E1 -18103.949,E2 -18103.949} C_VEL
LIN {X 0,Y 263.87,Z 505.199,A -85,B 0,C 180,E1 -18107.038,E2 -18107.038} C_VEL
LIN {X 0,Y 266.177,Z 498.432,A -85,B 0,C 180,E1 -18110.076,E2 -18110.076} C_VEL
LIN {X 0,Y 269.52,Z 490.27,A -85,B 0,C 180,E1 -18113.027,E2 -18113.027} C_VEL
LIN {X 0,Y 273.651,Z 480.625,A -85,B 0,C 180,E1 -18115.888,E2 -18115.888} C_VEL
LIN {X 0,Y 278.302,Z 470.795,A -85,B 0,C 180,E1 -18118.263,E2 -18118.263} C_VEL
LIN {X 0,Y 283.079,Z 458.143,A -85,B 0,C 180,E1 -18121.009,E2 -18121.009} C_VEL
LIN {X 0,Y 286.372,Z 448.392,A -85,B 0,C 180,E1 -18122.934,E2 -18122.934} C_VEL
LIN {X 0,Y 288.756,Z 438.826,A -85,B 0,C 180,E1 -18124.889,E2 -18124.889} C_VEL
LIN {X 0,Y 290.833,Z 428.275,A -85,B 0,C 180,E1 -18127.167,E2 -18127.167} C_VEL
LIN {X 0,Y 292.484,Z 417.708,A -85,B 0,C 180,E1 -18129.743,E2 -18129.743} C_VEL
LIN {X 0,Y 294.235,Z 407.6,A -85,B 0,C 180,E1 -18132.647,E2 -18132.647} C_VEL
LIN {X 0,Y 295.473,Z 402.299,A -85,B 0,C 180,E1 -18134.474,E2 -18134.474} C_VEL
LIN {X 0,Y 295.769,Z 400.493,A -85,B 0,C 180,E1 -18135.469,E2 -18135.469} C_VEL
LIN {X 0,Y 296,Z 398.556,A -85,B 0,C 180,E1 -18137.397,E2 -18137.397} C_VEL
LIN {X 0,Y 296.919,Z 397.281,A -85,B 0,C 180,E1 -18140.277,E2 -18140.277} C_VEL
LIN {X 0,Y 297.991,Z 397.297,A -85,B 0,C 180,E1 -18142.179,E2 -18142.179} C_VEL
LIN {X 0,Y 299.21,Z 398.16,A -85,B 0,C 180,E1 -18144.041,E2 -18144.041} C_VEL
LIN {X 0,Y 300.517,Z 399.735,A -85,B 0,C 180,E1 -18145.856,E2 -18145.856} C_VEL
LIN {X 0,Y 300.658,Z 402.626,A -85,B 0,C 180,E1 -18147.302,E2 -18147.302} C_VEL
LIN {X 0,Y 300.564,Z 404.703,A -85,B 0,C 180,E1 -18148.157,E2 -18148.157} C_VEL
LIN {X 0,Y 300.215,Z 405.988,A -85,B 0,C 180,E1 -18148.56,E2 -18148.56} C_VEL
LIN {X 0,Y 294.622,Z 416.372,A -85,B 0,C 180,E1 -18150.725,E2 -18150.725} C_VEL
LIN {X 0,Y 288.881,Z 425.924,A -85,B 0,C 180,E1 -18153.252,E2 -18153.252} C_VEL
LIN {X 0,Y 283.645,Z 433.769,A -85,B 0,C 180,E1 -18155.869,E2 -18155.869} C_VEL
LIN {X 0,Y 279.077,Z 440.065,A -85,B 0,C 180,E1 -18158.661,E2 -18158.661} C_VEL
LIN {X 0,Y 275.255,Z 444.676,A -85,B 0,C 180,E1 -18161.388,E2 -18161.388} C_VEL
LIN {X 0,Y 272.736,Z 447.378,A -85,B 0,C 180,E1 -18163.534,E2 -18163.534} C_VEL
LIN {X 0,Y 269.819,Z 449.875,A -85,B 0,C 180,E1 -18166.443,E2 -18166.443} C_VEL
LIN {X 0,Y 267.509,Z 451.107,A -85,B 0,C 180,E1 -18169.403,E2 -18169.403} C_VEL
LIN {X 0,Y 265.653,Z 451.12,A -85,B 0,C 180,E1 -18172.399,E2 -18172.399} C_VEL
LIN {X 0,Y 264.426,Z 449.853,A -85,B 0,C 180,E1 -18175.427,E2 -18175.427} C_VEL
LIN {X 0,Y 263.733,Z 447.3,A -85,B 0,C 180,E1 -18178.473,E2 -18178.473} C_VEL
LIN {X 0,Y 263.517,Z 443.426,A -85,B 0,C 180,E1 -18181.529,E2 -18181.529} C_VEL
LIN {X 0,Y 263.209,Z 438.183,A -85,B 0,C 180,E1 -18184.595,E2 -18184.595} C_VEL
LIN {X 0,Y 263.749,Z 433.182,A -85,B 0,C 180,E1 -18186.887,E2 -18186.887} C_VEL
LIN {X 0,Y 264.404,Z 425.653,A -85,B 0,C 180,E1 -18189.733,E2 -18189.733} C_VEL
LIN {X 0,Y 265.216,Z 417.589,A -85,B 0,C 180,E1 -18192.24,E2 -18192.24} C_VEL
LIN {X 0,Y 266.442,Z 407.228,A -85,B 0,C 180,E1 -18194.903,E2 -18194.903} C_VEL
LIN {X 0,Y 267.695,Z 396.521,A -85,B 0,C 180,E1 -18197.179,E2 -18197.179} C_VEL
LIN {X 0,Y 269.374,Z 383.72,A -85,B 0,C 180,E1 -18199.43,E2 -18199.43} C_VEL
LIN {X 0,Y 270.865,Z 370.823,A -85,B 0,C 180,E1 -18201.3,E2 -18201.3} C_VEL
LIN {X 0,Y 270.816,Z 367.958,A -85,B 0,C 180,E1 -18201.68,E2 -18201.68} C_VEL
LIN {X 0,Y 266.993,Z 354.135,A -85,B 0,C 180,E1 -18203.544,E2 -18203.544} C_VEL
LIN {X 0,Y 263.379,Z 340.994,A -85,B 0,C 180,E1 -18205.076,E2 -18205.076} C_VEL
LIN {X 0,Y 263.261,Z 340.35,A -85,B 0,C 180,E1 -18205.392,E2 -18205.392} C_VEL
LIN {X 0,Y 263.186,Z 340.328,A -85,B 0,C 180,E1 -18208.729,E2 -18208.729} C_VEL
LIN {X 0,Y 263.139,Z 340.333,A -85,B 0,C 180,E1 -18212.288,E2 -18212.288} C_VEL
LIN {X 0,Y 263.188,Z 340.325,A -85,B 0,C 180,E1 -18216.763,E2 -18216.763} C_VEL
LIN {X 0,Y 263.13,Z 340.331,A -85,B 0,C 180,E1 -18221.593,E2 -18221.593} C_VEL
LIN {X 0,Y 263.133,Z 340.33,A -85,B 0,C 180,E1 -18226.017,E2 -18226.017} C_VEL
LIN {X 0,Y 263.146,Z 340.332,A -85,B 0,C 180,E1 -18230.133,E2 -18230.133} C_VEL
LIN {X 0,Y 263.198,Z 340.323,A -85,B 0,C 180,E1 -18234.022,E2 -18234.022} C_VEL
LIN {X 0,Y 263.139,Z 340.331,A -85,B 0,C 180,E1 -18237.711,E2 -18237.711} C_VEL
LIN {X 0,Y 263.202,Z 340.323,A -85,B 0,C 180,E1 -18241.784,E2 -18241.784} C_VEL
LIN {X 0,Y 263.207,Z 340.321,A -85,B 0,C 180,E1 -18245.211,E2 -18245.211} C_VEL
LIN {X 0,Y 263.268,Z 340.315,A -85,B 0,C 180,E1 -18249.692,E2 -18249.692} C_VEL
LIN {X 0,Y 263.357,Z 340.304,A -85,B 0,C 180,E1 -18254.521,E2 -18254.521} C_VEL
LIN {X 0,Y 263.379,Z 340.299,A -85,B 0,C 180,E1 -18259.233,E2 -18259.233} C_VEL
LIN {X 0,Y 263.578,Z 340.276,A -85,B 0,C 180,E1 -18262.337,E2 -18262.337} C_VEL
LIN {X 0,Y 263.755,Z 340.252,A -85,B 0,C 180,E1 -18268.472,E2 -18268.472} C_VEL
LIN {X 0,Y 263.755,Z 340.256,A -85,B 0,C 180,E1 -18271.525,E2 -18271.525} C_VEL
LIN {X 0,Y 263.576,Z 340.279,A -85,B 0,C 180,E1 -18277.66,E2 -18277.66} C_VEL
LIN {X 0,Y 263.377,Z 340.3,A -85,B 0,C 180,E1 -18280.764,E2 -18280.764} C_VEL
LIN {X 0,Y 263.353,Z 340.305,A -85,B 0,C 180,E1 -18285.476,E2 -18285.476} C_VEL
LIN {X 0,Y 263.265,Z 340.314,A -85,B 0,C 180,E1 -18290.305,E2 -18290.305} C_VEL
LIN {X 0,Y 263.208,Z 340.324,A -85,B 0,C 180,E1 -18295.29,E2 -18295.29} C_VEL
LIN {X 0,Y 263.165,Z 340.327,A -85,B 0,C 180,E1 -18298.729,E2 -18298.729} C_VEL
LIN {X 0,Y 263.132,Z 340.329,A -85,B 0,C 180,E1 -18302.286,E2 -18302.286} C_VEL
LIN {X 0,Y 263.18,Z 340.326,A -85,B 0,C 180,E1 -18306.761,E2 -18306.761} C_VEL
LIN {X 0,Y 263.122,Z 340.332,A -85,B 0,C 180,E1 -18311.592,E2 -18311.592} C_VEL
LIN {X 0,Y 263.124,Z 340.331,A -85,B 0,C 180,E1 -18316.015,E2 -18316.015} C_VEL
LIN {X 0,Y 263.101,Z 340.333,A -85,B 0,C 180,E1 -18320.126,E2 -18320.126} C_VEL
LIN {X 0,Y 263.159,Z 340.327,A -85,B 0,C 180,E1 -18324.017,E2 -18324.017} C_VEL
LIN {X 0,Y 263.129,Z 340.329,A -85,B 0,C 180,E1 -18327.711,E2 -18327.711} C_VEL
LIN {X 0,Y 263.196,Z 340.323,A -85,B 0,C 180,E1 -18331.782,E2 -18331.782} C_VEL
LIN {X 0,Y 263.22,Z 340.319,A -85,B 0,C 180,E1 -18335.199,E2 -18335.199} C_VEL
LIN {X 0,Y 263.257,Z 340.315,A -85,B 0,C 180,E1 -18339.692,E2 -18339.692} C_VEL
LIN {X 0,Y 263.344,Z 340.307,A -85,B 0,C 180,E1 -18344.521,E2 -18344.521} C_VEL
LIN {X 0,Y 263.367,Z 340.302,A -85,B 0,C 180,E1 -18349.234,E2 -18349.234} C_VEL
LIN {X 0,Y 263.566,Z 340.279,A -85,B 0,C 180,E1 -18352.338,E2 -18352.338} C_VEL
LIN {X 0,Y 263.745,Z 340.258,A -85,B 0,C 180,E1 -18358.473,E2 -18358.473} C_VEL
LIN {X 0,Y 263.745,Z 340.253,A -85,B 0,C 180,E1 -18361.527,E2 -18361.527} C_VEL
LIN {X 0,Y 263.565,Z 340.277,A -85,B 0,C 180,E1 -18367.661,E2 -18367.661} C_VEL
LIN {X 0,Y 263.367,Z 340.301,A -85,B 0,C 180,E1 -18370.766,E2 -18370.766} C_VEL
LIN {X 0,Y 263.344,Z 340.305,A -85,B 0,C 180,E1 -18375.478,E2 -18375.478} C_VEL
LIN {X 0,Y 263.256,Z 340.318,A -85,B 0,C 180,E1 -18380.307,E2 -18380.307} C_VEL
LIN {X 0,Y 263.201,Z 340.322,A -85,B 0,C 180,E1 -18385.292,E2 -18385.292} C_VEL
LIN {X 0,Y 263.169,Z 340.325,A -85,B 0,C 180,E1 -18388.73,E2 -18388.73} C_VEL
LIN {X 0,Y 263.127,Z 340.334,A -85,B 0,C 180,E1 -18392.289,E2 -18392.289} C_VEL
LIN {X 0,Y 263.162,Z 340.33,A -85,B 0,C 180,E1 -18394.379,E2 -18394.379} C_VEL
LIN {X 0,Y 262.897,Z 340.717,A -85,B 0,C 180,E1 -18395.23,E2 -18395.23} C_VEL
LIN {X 0,Y 262.236,Z 341.704,A -85,B 0,C 180,E1 -18396.052,E2 -18396.052} C_VEL
LIN {X 0,Y 258.5,Z 347.775,A -85,B 0,C 180,E1 -18399.216,E2 -18399.216} C_VEL
LIN {X 0,Y 257.907,Z 350.063,A -85,B 0,C 180,E1 -18400.432,E2 -18400.432} C_VEL
LIN {X 0,Y 257.96,Z 350.797,A -85,B 0,C 180,E1 -18400.843,E2 -18400.843} C_VEL
LIN {X 0,Y 259.566,Z 358.804,A -85,B 0,C 180,E1 -18405.256,E2 -18405.256} C_VEL
LIN {X 0,Y 260.798,Z 364.685,A -85,B 0,C 180,E1 -18408.38,E2 -18408.38} C_VEL
LIN {X 0,Y 260.564,Z 367.234,A -85,B 0,C 180,E1 -18409.661,E2 -18409.661} C_VEL
LIN {X 0,Y 258.842,Z 376.118,A -85,B 0,C 180,E1 -18414.055,E2 -18414.055} C_VEL
LIN {X 0,Y 257.317,Z 385.651,A -85,B 0,C 180,E1 -18418.741,E2 -18418.741} C_VEL
LIN {X 0,Y 256.605,Z 390.901,A -85,B 0,C 180,E1 -18421.214,E2 -18421.214} C_VEL
LIN {X 0,Y 257.078,Z 399.497,A -85,B 0,C 180,E1 -18421.806,E2 -18421.806} C_VEL
LIN {X 0,Y 258.081,Z 414.779,A -85,B 0,C 180,E1 -18422.984,E2 -18422.984} C_VEL
LIN {X 0,Y 259.044,Z 430.023,A -85,B 0,C 180,E1 -18424.49,E2 -18424.49} C_VEL
LIN {X 0,Y 260.044,Z 444.584,A -85,B 0,C 180,E1 -18426.269,E2 -18426.269} C_VEL
LIN {X 0,Y 260.665,Z 455.262,A -85,B 0,C 180,E1 -18427.825,E2 -18427.825} C_VEL
LIN {X 0,Y 259.186,Z 466.685,A -85,B 0,C 180,E1 -18429.776,E2 -18429.776} C_VEL
LIN {X 0,Y 257.94,Z 476.286,A -85,B 0,C 180,E1 -18431.741,E2 -18431.741} C_VEL
LIN {X 0,Y 256.823,Z 485.973,A -85,B 0,C 180,E1 -18434.12,E2 -18434.12} C_VEL
LIN {X 0,Y 256.06,Z 495.26,A -85,B 0,C 180,E1 -18436.914,E2 -18436.914} C_VEL
LIN {X 0,Y 255.845,Z 502.753,A -85,B 0,C 180,E1 -18439.716,E2 -18439.716} C_VEL
LIN {X 0,Y 255.986,Z 507.901,A -85,B 0,C 180,E1 -18442.111,E2 -18442.111} C_VEL
LIN {X 0,Y 256.291,Z 511.984,A -85,B 0,C 180,E1 -18444.494,E2 -18444.494} C_VEL
LIN {X 0,Y 256.575,Z 515.005,A -85,B 0,C 180,E1 -18446.861,E2 -18446.861} C_VEL
LIN {X 0,Y 256.814,Z 516.494,A -85,B 0,C 180,E1 -18448.433,E2 -18448.433} C_VEL
LIN {X 0,Y 257.001,Z 517.562,A -85,B 0,C 180,E1 -18450.001,E2 -18450.001} C_VEL
LIN {X 0,Y 256.54,Z 518.103,A -85,B 0,C 180,E1 -18451.571,E2 -18451.571} C_VEL
LIN {X 0,Y 255.685,Z 518.083,A -85,B 0,C 180,E1 -18454.731,E2 -18454.731} C_VEL
LIN {X 0,Y 255.142,Z 516.953,A -85,B 0,C 180,E1 -18457.418,E2 -18457.418} C_VEL
LIN {X 0,Y 254.859,Z 515.449,A -85,B 0,C 180,E1 -18459.525,E2 -18459.525} C_VEL
LIN {X 0,Y 255.048,Z 512.089,A -85,B 0,C 180,E1 -18462.737,E2 -18462.737} C_VEL
LIN {X 0,Y 256.366,Z 506.787,A -85,B 0,C 180,E1 -18466.365,E2 -18466.365} C_VEL
LIN {X 0,Y 258.757,Z 500.003,A -85,B 0,C 180,E1 -18469.848,E2 -18469.848} C_VEL
LIN {X 0,Y 262,Z 492.538,A -85,B 0,C 180,E1 -18472.891,E2 -18472.891} C_VEL
LIN {X 0,Y 266.069,Z 483.92,A -85,B 0,C 180,E1 -18475.75,E2 -18475.75} C_VEL
LIN {X 0,Y 270.092,Z 476.032,A -85,B 0,C 180,E1 -18477.93,E2 -18477.93} C_VEL
LIN {X 0,Y 273.292,Z 468.98,A -85,B 0,C 180,E1 -18479.673,E2 -18479.673} C_VEL
LIN {X 0,Y 279.181,Z 454.936,A -85,B 0,C 180,E1 -18482.769,E2 -18482.769} C_VEL
LIN {X 0,Y 282.486,Z 444.891,A -85,B 0,C 180,E1 -18484.906,E2 -18484.906} C_VEL
LIN {X 0,Y 285.287,Z 434.133,A -85,B 0,C 180,E1 -18487.33,E2 -18487.33} C_VEL
LIN {X 0,Y 287.198,Z 425.33,A -85,B 0,C 180,E1 -18489.513,E2 -18489.513} C_VEL
LIN {X 0,Y 288.902,Z 417.538,A -85,B 0,C 180,E1 -18491.687,E2 -18491.687} C_VEL
LIN {X 0,Y 290.68,Z 410.548,A -85,B 0,C 180,E1 -18493.905,E2 -18493.905} C_VEL
LIN {X 0,Y 291.603,Z 407.413,A -85,B 0,C 180,E1 -18495.112,E2 -18495.112} C_VEL
LIN {X 0,Y 291.924,Z 405.708,A -85,B 0,C 180,E1 -18496.241,E2 -18496.241} C_VEL
LIN {X 0,Y 292.266,Z 404.057,A -85,B 0,C 180,E1 -18498.199,E2 -18498.199} C_VEL
LIN {X 0,Y 292.909,Z 403.231,A -85,B 0,C 180,E1 -18500.158,E2 -18500.158} C_VEL
LIN {X 0,Y 293.885,Z 403.122,A -85,B 0,C 180,E1 -18502.109,E2 -18502.109} C_VEL
LIN {X 0,Y 295.014,Z 403.916,A -85,B 0,C 180,E1 -18504.094,E2 -18504.094} C_VEL
LIN {X 0,Y 295.687,Z 404.751,A -85,B 0,C 180,E1 -18505.219,E2 -18505.219} C_VEL
LIN {X 0,Y 296.019,Z 406.029,A -85,B 0,C 180,E1 -18506.199,E2 -18506.199} C_VEL
LIN {X 0,Y 295.705,Z 408.929,A -85,B 0,C 180,E1 -18507.57,E2 -18507.57} C_VEL
LIN {X 0,Y 294.053,Z 412.077,A -85,B 0,C 180,E1 -18508.277,E2 -18508.277} C_VEL
LIN {X 0,Y 288.421,Z 421.381,A -85,B 0,C 180,E1 -18510.434,E2 -18510.434} C_VEL
LIN {X 0,Y 283.168,Z 429.234,A -85,B 0,C 180,E1 -18512.668,E2 -18512.668} C_VEL
LIN {X 0,Y 277.682,Z 436.624,A -85,B 0,C 180,E1 -18515.317,E2 -18515.317} C_VEL
LIN {X 0,Y 272.984,Z 442.405,A -85,B 0,C 180,E1 -18518.081,E2 -18518.081} C_VEL
LIN {X 0,Y 269.824,Z 445.89,A -85,B 0,C 180,E1 -18520.208,E2 -18520.208} C_VEL
LIN {X 0,Y 266.206,Z 449.336,A -85,B 0,C 180,E1 -18523.118,E2 -18523.118} C_VEL
LIN {X 0,Y 263.139,Z 451.555,A -85,B 0,C 180,E1 -18526.092,E2 -18526.092} C_VEL
LIN {X 0,Y 260.698,Z 452.549,A -85,B 0,C 180,E1 -18529.123,E2 -18529.123} C_VEL
LIN {X 0,Y 258.722,Z 452.346,A -85,B 0,C 180,E1 -18532.194,E2 -18532.194} C_VEL
LIN {X 0,Y 257.43,Z 450.865,A -85,B 0,C 180,E1 -18535.303,E2 -18535.303} C_VEL
LIN {X 0,Y 256.689,Z 448.109,A -85,B 0,C 180,E1 -18538.431,E2 -18538.431} C_VEL
LIN {X 0,Y 256.443,Z 444.038,A -85,B 0,C 180,E1 -18541.571,E2 -18541.571} C_VEL
LIN {X 0,Y 256.152,Z 438.587,A -85,B 0,C 180,E1 -18544.722,E2 -18544.722} C_VEL
LIN {X 0,Y 256.716,Z 433.398,A -85,B 0,C 180,E1 -18547.077,E2 -18547.077} C_VEL
LIN {X 0,Y 257.367,Z 425.899,A -85,B 0,C 180,E1 -18549.919,E2 -18549.919} C_VEL
LIN {X 0,Y 258.241,Z 417.363,A -85,B 0,C 180,E1 -18552.576,E2 -18552.576} C_VEL
LIN {X 0,Y 259.528,Z 406.672,A -85,B 0,C 180,E1 -18555.31,E2 -18555.31} C_VEL
LIN {X 0,Y 260.863,Z 395.701,A -85,B 0,C 180,E1 -18557.644,E2 -18557.644} C_VEL
LIN {X 0,Y 262.463,Z 383.729,A -85,B 0,C 180,E1 -18559.759,E2 -18559.759} C_VEL
LIN {X 0,Y 264.001,Z 370.292,A -85,B 0,C 180,E1 -18561.72,E2 -18561.72} C_VEL
LIN {X 0,Y 260.586,Z 357.548,A -85,B 0,C 180,E1 -18563.509,E2 -18563.509} C_VEL
LIN {X 0,Y 256.318,Z 341.756,A -85,B 0,C 180,E1 -18565.447,E2 -18565.447} C_VEL
LIN {X 0,Y 256.219,Z 341.217,A -85,B 0,C 180,E1 -18565.779,E2 -18565.779} C_VEL
LIN {X 0,Y 256.12,Z 341.206,A -85,B 0,C 180,E1 -18569.599,E2 -18569.599} C_VEL
LIN {X 0,Y 256.073,Z 341.211,A -85,B 0,C 180,E1 -18573.293,E2 -18573.293} C_VEL
LIN {X 0,Y 256.12,Z 341.203,A -85,B 0,C 180,E1 -18577.271,E2 -18577.271} C_VEL
LIN {X 0,Y 256.06,Z 341.212,A -85,B 0,C 180,E1 -18581.203,E2 -18581.203} C_VEL
LIN {X 0,Y 256.067,Z 341.209,A -85,B 0,C 180,E1 -18585.529,E2 -18585.529} C_VEL
LIN {X 0,Y 256.091,Z 341.209,A -85,B 0,C 180,E1 -18588.802,E2 -18588.802} C_VEL
LIN {X 0,Y 256.161,Z 341.198,A -85,B 0,C 180,E1 -18592.871,E2 -18592.871} C_VEL
LIN {X 0,Y 256.091,Z 341.209,A -85,B 0,C 180,E1 -18596.709,E2 -18596.709} C_VEL
LIN {X 0,Y 256.132,Z 341.202,A -85,B 0,C 180,E1 -18601.409,E2 -18601.409} C_VEL
LIN {X 0,Y 256.148,Z 341.202,A -85,B 0,C 180,E1 -18605.696,E2 -18605.696} C_VEL
LIN {X 0,Y 256.168,Z 341.197,A -85,B 0,C 180,E1 -18609.104,E2 -18609.104} C_VEL
LIN {X 0,Y 256.306,Z 341.185,A -85,B 0,C 180,E1 -18614.084,E2 -18614.084} C_VEL
LIN {X 0,Y 256.315,Z 341.178,A -85,B 0,C 180,E1 -18618.933,E2 -18618.933} C_VEL
LIN {X 0,Y 256.545,Z 341.154,A -85,B 0,C 180,E1 -18622.126,E2 -18622.126} C_VEL
LIN {X 0,Y 256.718,Z 341.129,A -85,B 0,C 180,E1 -18628.43,E2 -18628.43} C_VEL
LIN {X 0,Y 256.718,Z 341.133,A -85,B 0,C 180,E1 -18631.567,E2 -18631.567} C_VEL
LIN {X 0,Y 256.544,Z 341.154,A -85,B 0,C 180,E1 -18637.871,E2 -18637.871} C_VEL
LIN {X 0,Y 256.313,Z 341.181,A -85,B 0,C 180,E1 -18641.064,E2 -18641.064} C_VEL
LIN {X 0,Y 256.302,Z 341.182,A -85,B 0,C 180,E1 -18645.913,E2 -18645.913} C_VEL
LIN {X 0,Y 256.169,Z 341.199,A -85,B 0,C 180,E1 -18650.893,E2 -18650.893} C_VEL
LIN {X 0,Y 256.188,Z 341.197,A -85,B 0,C 180,E1 -18655.137,E2 -18655.137} C_VEL
LIN {X 0,Y 256.103,Z 341.208,A -85,B 0,C 180,E1 -18659.599,E2 -18659.599} C_VEL
LIN {X 0,Y 256.066,Z 341.214,A -85,B 0,C 180,E1 -18663.291,E2 -18663.291} C_VEL
LIN {X 0,Y 256.112,Z 341.209,A -85,B 0,C 180,E1 -18667.269,E2 -18667.269} C_VEL
LIN {X 0,Y 256.053,Z 341.215,A -85,B 0,C 180,E1 -18671.202,E2 -18671.202} C_VEL
LIN {X 0,Y 256.059,Z 341.213,A -85,B 0,C 180,E1 -18675.527,E2 -18675.527} C_VEL
LIN {X 0,Y 256.051,Z 341.214,A -85,B 0,C 180,E1 -18678.795,E2 -18678.795} C_VEL
LIN {X 0,Y 256.126,Z 341.207,A -85,B 0,C 180,E1 -18682.866,E2 -18682.866} C_VEL
LIN {X 0,Y 256.063,Z 341.214,A -85,B 0,C 180,E1 -18686.706,E2 -18686.706} C_VEL
LIN {X 0,Y 256.109,Z 341.207,A -85,B 0,C 180,E1 -18690.399,E2 -18690.399} C_VEL
LIN {X 0,Y 256.183,Z 341.198,A -85,B 0,C 180,E1 -18694.86,E2 -18694.86} C_VEL
LIN {X 0,Y 256.161,Z 341.201,A -85,B 0,C 180,E1 -18699.104,E2 -18699.104} C_VEL
LIN {X 0,Y 256.293,Z 341.182,A -85,B 0,C 180,E1 -18704.084,E2 -18704.084} C_VEL
LIN {X 0,Y 256.303,Z 341.183,A -85,B 0,C 180,E1 -18708.933,E2 -18708.933} C_VEL
LIN {X 0,Y 256.534,Z 341.154,A -85,B 0,C 180,E1 -18712.126,E2 -18712.126} C_VEL
LIN {X 0,Y 256.708,Z 341.135,A -85,B 0,C 180,E1 -18718.431,E2 -18718.431} C_VEL
LIN {X 0,Y 256.708,Z 341.129,A -85,B 0,C 180,E1 -18721.568,E2 -18721.568} C_VEL
LIN {X 0,Y 256.533,Z 341.154,A -85,B 0,C 180,E1 -18727.873,E2 -18727.873} C_VEL
LIN {X 0,Y 256.303,Z 341.18,A -85,B 0,C 180,E1 -18731.066,E2 -18731.066} C_VEL
LIN {X 0,Y 256.293,Z 341.186,A -85,B 0,C 180,E1 -18735.915,E2 -18735.915} C_VEL
LIN {X 0,Y 256.159,Z 341.199,A -85,B 0,C 180,E1 -18740.895,E2 -18740.895} C_VEL
LIN {X 0,Y 256.181,Z 341.196,A -85,B 0,C 180,E1 -18745.139,E2 -18745.139} C_VEL
LIN {X 0,Y 256.104,Z 341.207,A -85,B 0,C 180,E1 -18749.6,E2 -18749.6} C_VEL
LIN {X 0,Y 256.129,Z 341.207,A -85,B 0,C 180,E1 -18754.599,E2 -18754.599} C_VEL
LIN {X 0,Y 256.213,Z 341.48,A -85,B 0,C 180,E1 -18755.413,E2 -18755.413} C_VEL
LIN {X 0,Y 257.766,Z 349.73,A -85,B 0,C 180,E1 -18760.236,E2 -18760.236} C_VEL
LIN {X 0,Y 257.96,Z 350.797,A -85,B 0,C 180,E1 -18760.843,E2 -18760.843} C_VEL
LIN {X 0,Y 257.696,Z 353.061,A -85,B 0,C 180,E1 -18762.054,E2 -18762.054} C_VEL
LIN {X 0,Y 255.551,Z 357.008,A -85,B 0,C 180,E1 -18764.029,E2 -18764.029} C_VEL
LIN {X 0,Y 253.466,Z 361.006,A -85,B 0,C 180,E1 -18766.035,E2 -18766.035} C_VEL
LIN {X 0,Y 253.324,Z 363.345,A -85,B 0,C 180,E1 -18767.273,E2 -18767.273} C_VEL
LIN {X 0,Y 253.727,Z 365.451,A -85,B 0,C 180,E1 -18768.406,E2 -18768.406} C_VEL
LIN {X 0,Y 253.191,Z 369.167,A -85,B 0,C 180,E1 -18770.328,E2 -18770.328} C_VEL
LIN {X 0,Y 251.345,Z 378.387,A -85,B 0,C 180,E1 -18775.028,E2 -18775.028} C_VEL
LIN {X 0,Y 249.934,Z 387.385,A -85,B 0,C 180,E1 -18779.594,E2 -18779.594} C_VEL
LIN {X 0,Y 249.591,Z 390.059,A -85,B 0,C 180,E1 -18780.818,E2 -18780.818} C_VEL
LIN {X 0,Y 250.721,Z 409.941,A -85,B 0,C 180,E1 -18782.294,E2 -18782.294} C_VEL
LIN {X 0,Y 251.74,Z 425.546,A -85,B 0,C 180,E1 -18783.793,E2 -18783.793} C_VEL
LIN {X 0,Y 252.601,Z 439.63,A -85,B 0,C 180,E1 -18785.485,E2 -18785.485} C_VEL
LIN {X 0,Y 253.442,Z 452.689,A -85,B 0,C 180,E1 -18787.373,E2 -18787.373} C_VEL
LIN {X 0,Y 253.434,Z 456.663,A -85,B 0,C 180,E1 -18788.016,E2 -18788.016} C_VEL
LIN {X 0,Y 251.823,Z 468.606,A -85,B 0,C 180,E1 -18790.223,E2 -18790.223} C_VEL
LIN {X 0,Y 250.509,Z 478.122,A -85,B 0,C 180,E1 -18792.346,E2 -18792.346} C_VEL
LIN {X 0,Y 249.512,Z 487.663,A -85,B 0,C 180,E1 -18794.899,E2 -18794.899} C_VEL
LIN {X 0,Y 248.939,Z 496.43,A -85,B 0,C 180,E1 -18797.777,E2 -18797.777} C_VEL
LIN {X 0,Y 248.884,Z 502.547,A -85,B 0,C 180,E1 -18800.247,E2 -18800.247} C_VEL
LIN {X 0,Y 249.077,Z 507.469,A -85,B 0,C 180,E1 -18802.707,E2 -18802.707} C_VEL
LIN {X 0,Y 249.458,Z 511.343,A -85,B 0,C 180,E1 -18805.153,E2 -18805.153} C_VEL
LIN {X 0,Y 249.634,Z 513.334,A -85,B 0,C 180,E1 -18806.774,E2 -18806.774} C_VEL
LIN {X 0,Y 249.868,Z 514.907,A -85,B 0,C 180,E1 -18808.39,E2 -18808.39} C_VEL
LIN {X 0,Y 250.071,Z 516.057,A -85,B 0,C 180,E1 -18810.001,E2 -18810.001} C_VEL
LIN {X 0,Y 249.076,Z 516.903,A -85,B 0,C 180,E1 -18813.237,E2 -18813.237} C_VEL
LIN {X 0,Y 248.342,Z 516.342,A -85,B 0,C 180,E1 -18816.501,E2 -18816.501} C_VEL
LIN {X 0,Y 247.8,Z 514.413,A -85,B 0,C 180,E1 -18819.799,E2 -18819.799} C_VEL
LIN {X 0,Y 248.044,Z 511.259,A -85,B 0,C 180,E1 -18823.102,E2 -18823.102} C_VEL
LIN {X 0,Y 249.366,Z 506.542,A -85,B 0,C 180,E1 -18826.618,E2 -18826.618} C_VEL
LIN {X 0,Y 251.331,Z 501.343,A -85,B 0,C 180,E1 -18829.608,E2 -18829.608} C_VEL
LIN {X 0,Y 254.461,Z 494.531,A -85,B 0,C 180,E1 -18832.749,E2 -18832.749} C_VEL
LIN {X 0,Y 259.25,Z 485.287,A -85,B 0,C 180,E1 -18836.138,E2 -18836.138} C_VEL
LIN {X 0,Y 261.784,Z 480.499,A -85,B 0,C 180,E1 -18837.634,E2 -18837.634} C_VEL
LIN {X 0,Y 266.028,Z 472.9,A -85,B 0,C 180,E1 -18839.694,E2 -18839.694} C_VEL
LIN {X 0,Y 271.344,Z 461.472,A -85,B 0,C 180,E1 -18842.511,E2 -18842.511} C_VEL
LIN {X 0,Y 275.323,Z 452.258,A -85,B 0,C 180,E1 -18844.574,E2 -18844.574} C_VEL
LIN {X 0,Y 279.114,Z 441.014,A -85,B 0,C 180,E1 -18847.181,E2 -18847.181} C_VEL
LIN {X 0,Y 282.052,Z 430.761,A -85,B 0,C 180,E1 -18849.792,E2 -18849.792} C_VEL
LIN {X 0,Y 284.555,Z 421.605,A -85,B 0,C 180,E1 -18852.469,E2 -18852.469} C_VEL
LIN {X 0,Y 286.696,Z 414.984,A -85,B 0,C 180,E1 -18854.692,E2 -18854.692} C_VEL
LIN {X 0,Y 287.695,Z 412.165,A -85,B 0,C 180,E1 -18855.898,E2 -18855.898} C_VEL
LIN {X 0,Y 287.939,Z 410.807,A -85,B 0,C 180,E1 -18857.076,E2 -18857.076} C_VEL
LIN {X 0,Y 288.379,Z 409.444,A -85,B 0,C 180,E1 -18859.07,E2 -18859.07} C_VEL
LIN {X 0,Y 289.123,Z 408.864,A -85,B 0,C 180,E1 -18861.066,E2 -18861.066} C_VEL
LIN {X 0,Y 290.08,Z 409.045,A -85,B 0,C 180,E1 -18863.085,E2 -18863.085} C_VEL
LIN {X 0,Y 291.129,Z 410.218,A -85,B 0,C 180,E1 -18865.164,E2 -18865.164} C_VEL
LIN {X 0,Y 291.146,Z 411.816,A -85,B 0,C 180,E1 -18866.276,E2 -18866.276} C_VEL
LIN {X 0,Y 291,Z 412.627,A -85,B 0,C 180,E1 -18866.682,E2 -18866.682} C_VEL
LIN {X 0,Y 290.162,Z 414.288,A -85,B 0,C 180,E1 -18867.189,E2 -18867.189} C_VEL
LIN {X 0,Y 283.789,Z 423.985,A -85,B 0,C 180,E1 -18869.491,E2 -18869.491} C_VEL
LIN {X 0,Y 277.495,Z 432.506,A -85,B 0,C 180,E1 -18872.061,E2 -18872.061} C_VEL
LIN {X 0,Y 271.747,Z 439.479,A -85,B 0,C 180,E1 -18874.74,E2 -18874.74} C_VEL
LIN {X 0,Y 266.406,Z 445.348,A -85,B 0,C 180,E1 -18877.8,E2 -18877.8} C_VEL
LIN {X 0,Y 261.496,Z 449.858,A -85,B 0,C 180,E1 -18881.185,E2 -18881.185} C_VEL
LIN {X 0,Y 257.99,Z 452.415,A -85,B 0,C 180,E1 -18884.192,E2 -18884.192} C_VEL
LIN {X 0,Y 255.09,Z 453.771,A -85,B 0,C 180,E1 -18887.267,E2 -18887.267} C_VEL
LIN {X 0,Y 252.784,Z 453.93,A -85,B 0,C 180,E1 -18890.398,E2 -18890.398} C_VEL
LIN {X 0,Y 251.031,Z 452.873,A -85,B 0,C 180,E1 -18893.571,E2 -18893.571} C_VEL
LIN {X 0,Y 249.994,Z 450.538,A -85,B 0,C 180,E1 -18896.777,E2 -18896.777} C_VEL
LIN {X 0,Y 249.5,Z 446.917,A -85,B 0,C 180,E1 -18900,E2 -18900} C_VEL
LIN {X 0,Y 249.24,Z 443.295,A -85,B 0,C 180,E1 -18902.425,E2 -18902.425} C_VEL
LIN {X 0,Y 249.279,Z 437.213,A -85,B 0,C 180,E1 -18905.663,E2 -18905.663} C_VEL
LIN {X 0,Y 249.878,Z 430.534,A -85,B 0,C 180,E1 -18908.492,E2 -18908.492} C_VEL
LIN {X 0,Y 250.669,Z 422.4,A -85,B 0,C 180,E1 -18911.319,E2 -18911.319} C_VEL
LIN {X 0,Y 251.808,Z 412.554,A -85,B 0,C 180,E1 -18914.136,E2 -18914.136} C_VEL
LIN {X 0,Y 253.035,Z 402.481,A -85,B 0,C 180,E1 -18916.541,E2 -18916.541} C_VEL
LIN {X 0,Y 254.611,Z 390.509,A -85,B 0,C 180,E1 -18918.926,E2 -18918.926} C_VEL
LIN {X 0,Y 256.26,Z 377.823,A -85,B 0,C 180,E1 -18921.013,E2 -18921.013} C_VEL
LIN {X 0,Y 257,Z 371.442,A -85,B 0,C 180,E1 -18921.923,E2 -18921.923} C_VEL
LIN {X 0,Y 253.503,Z 358.329,A -85,B 0,C 180,E1 -18923.809,E2 -18923.809} C_VEL
LIN {X 0,Y 249.272,Z 342.667,A -85,B 0,C 180,E1 -18925.773,E2 -18925.773} C_VEL
LIN {X 0,Y 249.15,Z 342.104,A -85,B 0,C 180,E1 -18926.103,E2 -18926.103} C_VEL
LIN {X 0,Y 249.058,Z 342.088,A -85,B 0,C 180,E1 -18930.527,E2 -18930.527} C_VEL
LIN {X 0,Y 249.051,Z 342.086,A -85,B 0,C 180,E1 -18935.078,E2 -18935.078} C_VEL
LIN {X 0,Y 249.031,Z 342.089,A -85,B 0,C 180,E1 -18938.38,E2 -18938.38} C_VEL
LIN {X 0,Y 249.015,Z 342.09,A -85,B 0,C 180,E1 -18942.792,E2 -18942.792} C_VEL
LIN {X 0,Y 249.036,Z 342.086,A -85,B 0,C 180,E1 -18947.365,E2 -18947.365} C_VEL
LIN {X 0,Y 249.054,Z 342.084,A -85,B 0,C 180,E1 -18951.623,E2 -18951.623} C_VEL
LIN {X 0,Y 249.068,Z 342.082,A -85,B 0,C 180,E1 -18955.642,E2 -18955.642} C_VEL
LIN {X 0,Y 249.053,Z 342.085,A -85,B 0,C 180,E1 -18959.472,E2 -18959.472} C_VEL
LIN {X 0,Y 249.074,Z 342.08,A -85,B 0,C 180,E1 -18963.161,E2 -18963.161} C_VEL
LIN {X 0,Y 249.067,Z 342.083,A -85,B 0,C 180,E1 -18966.73,E2 -18966.73} C_VEL
LIN {X 0,Y 249.115,Z 342.078,A -85,B 0,C 180,E1 -18970.211,E2 -18970.211} C_VEL
LIN {X 0,Y 249.247,Z 342.062,A -85,B 0,C 180,E1 -18973.621,E2 -18973.621} C_VEL
LIN {X 0,Y 249.258,Z 342.057,A -85,B 0,C 180,E1 -18978.615,E2 -18978.615} C_VEL
LIN {X 0,Y 249.489,Z 342.034,A -85,B 0,C 180,E1 -18981.902,E2 -18981.902} C_VEL
LIN {X 0,Y 249.441,Z 342.035,A -85,B 0,C 180,E1 -18986.768,E2 -18986.768} C_VEL
LIN {X 0,Y 249.732,Z 342.002,A -85,B 0,C 180,E1 -18989.999,E2 -18989.999} C_VEL
LIN {X 0,Y 249.44,Z 342.038,A -85,B 0,C 180,E1 -18993.229,E2 -18993.229} C_VEL
LIN {X 0,Y 249.488,Z 342.031,A -85,B 0,C 180,E1 -18998.095,E2 -18998.095} C_VEL
LIN {X 0,Y 249.256,Z 342.062,A -85,B 0,C 180,E1 -19001.382,E2 -19001.382} C_VEL
LIN {X 0,Y 249.244,Z 342.06,A -85,B 0,C 180,E1 -19006.376,E2 -19006.376} C_VEL
LIN {X 0,Y 249.088,Z 342.082,A -85,B 0,C 180,E1 -19011.516,E2 -19011.516} C_VEL
LIN {X 0,Y 249.131,Z 342.078,A -85,B 0,C 180,E1 -19015.48,E2 -19015.48} C_VEL
LIN {X 0,Y 249.073,Z 342.084,A -85,B 0,C 180,E1 -19018.987,E2 -19018.987} C_VEL
LIN {X 0,Y 249.029,Z 342.085,A -85,B 0,C 180,E1 -19022.424,E2 -19022.424} C_VEL
LIN {X 0,Y 249.028,Z 342.088,A -85,B 0,C 180,E1 -19026.344,E2 -19026.344} C_VEL
LIN {X 0,Y 249.004,Z 342.089,A -85,B 0,C 180,E1 -19030.476,E2 -19030.476} C_VEL
LIN {X 0,Y 249.004,Z 342.094,A -85,B 0,C 180,E1 -19034.876,E2 -19034.876} C_VEL
LIN {X 0,Y 249.015,Z 342.09,A -85,B 0,C 180,E1 -19037.362,E2 -19037.362} C_VEL
LIN {X 0,Y 249.04,Z 342.086,A -85,B 0,C 180,E1 -19042.198,E2 -19042.198} C_VEL
LIN {X 0,Y 249.039,Z 342.086,A -85,B 0,C 180,E1 -19045.638,E2 -19045.638} C_VEL
LIN {X 0,Y 249.047,Z 342.085,A -85,B 0,C 180,E1 -19049.472,E2 -19049.472} C_VEL
LIN {X 0,Y 249.069,Z 342.084,A -85,B 0,C 180,E1 -19053.161,E2 -19053.161} C_VEL
LIN {X 0,Y 249.074,Z 342.084,A -85,B 0,C 180,E1 -19056.732,E2 -19056.732} C_VEL
LIN {X 0,Y 249.105,Z 342.079,A -85,B 0,C 180,E1 -19060.211,E2 -19060.211} C_VEL
LIN {X 0,Y 249.236,Z 342.06,A -85,B 0,C 180,E1 -19063.621,E2 -19063.621} C_VEL
LIN {X 0,Y 249.246,Z 342.065,A -85,B 0,C 180,E1 -19068.616,E2 -19068.616} C_VEL
LIN {X 0,Y 249.478,Z 342.032,A -85,B 0,C 180,E1 -19071.902,E2 -19071.902} C_VEL
LIN {X 0,Y 249.431,Z 342.04,A -85,B 0,C 180,E1 -19076.769,E2 -19076.769} C_VEL
LIN {X 0,Y 249.721,Z 342.003,A -85,B 0,C 180,E1 -19080,E2 -19080} C_VEL
LIN {X 0,Y 249.431,Z 342.036,A -85,B 0,C 180,E1 -19083.23,E2 -19083.23} C_VEL
LIN {X 0,Y 249.477,Z 342.035,A -85,B 0,C 180,E1 -19088.097,E2 -19088.097} C_VEL
LIN {X 0,Y 249.246,Z 342.059,A -85,B 0,C 180,E1 -19091.383,E2 -19091.383} C_VEL
LIN {X 0,Y 249.235,Z 342.064,A -85,B 0,C 180,E1 -19096.378,E2 -19096.378} C_VEL
LIN {X 0,Y 249.08,Z 342.082,A -85,B 0,C 180,E1 -19101.518,E2 -19101.518} C_VEL
LIN {X 0,Y 249.124,Z 342.076,A -85,B 0,C 180,E1 -19105.483,E2 -19105.483} C_VEL
LIN {X 0,Y 249.074,Z 342.081,A -85,B 0,C 180,E1 -19108.993,E2 -19108.993} C_VEL
LIN {X 0,Y 249.03,Z 342.09,A -85,B 0,C 180,E1 -19112.426,E2 -19112.426} C_VEL
LIN {X 0,Y 249.129,Z 342.297,A -85,B 0,C 180,E1 -19115.108,E2 -19115.108} C_VEL
LIN {X 0,Y 250.407,Z 348.999,A -85,B 0,C 180,E1 -19119.16,E2 -19119.16} C_VEL
LIN {X 0,Y 252.138,Z 357.703,A -85,B 0,C 180,E1 -19124.174,E2 -19124.174} C_VEL
LIN {X 0,Y 253.324,Z 363.345,A -85,B 0,C 180,E1 -19127.273,E2 -19127.273} C_VEL
LIN {X 0,Y 253.242,Z 364.888,A -85,B 0,C 180,E1 -19128.085,E2 -19128.085} C_VEL
LIN {X 0,Y 251.894,Z 367.266,A -85,B 0,C 180,E1 -19129.273,E2 -19129.273} C_VEL
LIN {X 0,Y 245.408,Z 374.428,A -85,B 0,C 180,E1 -19132.821,E2 -19132.821} C_VEL
LIN {X 0,Y 244.739,Z 376.058,A -85,B 0,C 180,E1 -19133.672,E2 -19133.672} C_VEL
LIN {X 0,Y 243.144,Z 385.532,A -85,B 0,C 180,E1 -19138.651,E2 -19138.651} C_VEL
LIN {X 0,Y 242.616,Z 389.255,A -85,B 0,C 180,E1 -19140.429,E2 -19140.429} C_VEL
LIN {X 0,Y 243.522,Z 407.521,A -85,B 0,C 180,E1 -19141.8,E2 -19141.8} C_VEL
LIN {X 0,Y 244.511,Z 422.984,A -85,B 0,C 180,E1 -19143.305,E2 -19143.305} C_VEL
LIN {X 0,Y 245.342,Z 437.198,A -85,B 0,C 180,E1 -19145.026,E2 -19145.026} C_VEL
LIN {X 0,Y 246.271,Z 451.358,A -85,B 0,C 180,E1 -19147.12,E2 -19147.12} C_VEL
LIN {X 0,Y 246.308,Z 456.638,A -85,B 0,C 180,E1 -19148.008,E2 -19148.008} C_VEL
LIN {X 0,Y 244.715,Z 468.411,A -85,B 0,C 180,E1 -19150.28,E2 -19150.28} C_VEL
LIN {X 0,Y 243.295,Z 478.609,A -85,B 0,C 180,E1 -19152.679,E2 -19152.679} C_VEL
LIN {X 0,Y 242.392,Z 487.825,A -85,B 0,C 180,E1 -19155.305,E2 -19155.305} C_VEL
LIN {X 0,Y 241.888,Z 496.27,A -85,B 0,C 180,E1 -19158.267,E2 -19158.267} C_VEL
LIN {X 0,Y 241.952,Z 502.528,A -85,B 0,C 180,E1 -19160.967,E2 -19160.967} C_VEL
LIN {X 0,Y 242.18,Z 506.973,A -85,B 0,C 180,E1 -19163.336,E2 -19163.336} C_VEL
LIN {X 0,Y 242.581,Z 510.633,A -85,B 0,C 180,E1 -19165.848,E2 -19165.848} C_VEL
LIN {X 0,Y 242.913,Z 513.293,A -85,B 0,C 180,E1 -19168.344,E2 -19168.344} C_VEL
LIN {X 0,Y 243.124,Z 514.528,A -85,B 0,C 180,E1 -19170.002,E2 -19170.002} C_VEL
LIN {X 0,Y 242.588,Z 515.207,A -85,B 0,C 180,E1 -19171.662,E2 -19171.662} C_VEL
LIN {X 0,Y 241.615,Z 515.487,A -85,B 0,C 180,E1 -19175.008,E2 -19175.008} C_VEL
LIN {X 0,Y 241.056,Z 514.788,A -85,B 0,C 180,E1 -19177.577,E2 -19177.577} C_VEL
LIN {X 0,Y 240.735,Z 513.383,A -85,B 0,C 180,E1 -19180.09,E2 -19180.09} C_VEL
LIN {X 0,Y 241.056,Z 510.448,A -85,B 0,C 180,E1 -19183.489,E2 -19183.489} C_VEL
LIN {X 0,Y 242.386,Z 506.282,A -85,B 0,C 180,E1 -19186.896,E2 -19186.896} C_VEL
LIN {X 0,Y 244.596,Z 501.028,A -85,B 0,C 180,E1 -19190.171,E2 -19190.171} C_VEL
LIN {X 0,Y 247.916,Z 494.533,A -85,B 0,C 180,E1 -19193.384,E2 -19193.384} C_VEL
LIN {X 0,Y 252.907,Z 485.751,A -85,B 0,C 180,E1 -19196.846,E2 -19196.846} C_VEL
LIN {X 0,Y 256.249,Z 480.111,A -85,B 0,C 180,E1 -19198.683,E2 -19198.683} C_VEL
LIN {X 0,Y 260.585,Z 472.663,A -85,B 0,C 180,E1 -19200.827,E2 -19200.827} C_VEL
LIN {X 0,Y 266.315,Z 461.674,A -85,B 0,C 180,E1 -19203.656,E2 -19203.656} C_VEL
LIN {X 0,Y 269.946,Z 453.945,A -85,B 0,C 180,E1 -19205.494,E2 -19205.494} C_VEL
LIN {X 0,Y 273.945,Z 443.792,A -85,B 0,C 180,E1 -19208.005,E2 -19208.005} C_VEL
LIN {X 0,Y 277.099,Z 434.684,A -85,B 0,C 180,E1 -19210.458,E2 -19210.458} C_VEL
LIN {X 0,Y 280.216,Z 425.408,A -85,B 0,C 180,E1 -19213.336,E2 -19213.336} C_VEL
LIN {X 0,Y 282.313,Z 420.075,A -85,B 0,C 180,E1 -19215.198,E2 -19215.198} C_VEL
LIN {X 0,Y 283.17,Z 418.075,A -85,B 0,C 180,E1 -19216.035,E2 -19216.035} C_VEL
LIN {X 0,Y 283.552,Z 416.887,A -85,B 0,C 180,E1 -19216.83,E2 -19216.83} C_VEL
LIN {X 0,Y 283.787,Z 415.828,A -85,B 0,C 180,E1 -19218.037,E2 -19218.037} C_VEL
LIN {X 0,Y 284.315,Z 414.776,A -85,B 0,C 180,E1 -19220.023,E2 -19220.023} C_VEL
LIN {X 0,Y 285.118,Z 414.438,A -85,B 0,C 180,E1 -19222.073,E2 -19222.073} C_VEL
LIN {X 0,Y 286.023,Z 414.988,A -85,B 0,C 180,E1 -19224.181,E2 -19224.181} C_VEL
LIN {X 0,Y 286.29,Z 416.271,A -85,B 0,C 180,E1 -19225.625,E2 -19225.625} C_VEL
LIN {X 0,Y 285.516,Z 418.033,A -85,B 0,C 180,E1 -19226.369,E2 -19226.369} C_VEL
LIN {X 0,Y 279.275,Z 426.659,A -85,B 0,C 180,E1 -19228.522,E2 -19228.522} C_VEL
LIN {X 0,Y 273.427,Z 433.952,A -85,B 0,C 180,E1 -19230.767,E2 -19230.767} C_VEL
LIN {X 0,Y 267.289,Z 440.832,A -85,B 0,C 180,E1 -19233.45,E2 -19233.45} C_VEL
LIN {X 0,Y 261.938,Z 446.248,A -85,B 0,C 180,E1 -19236.268,E2 -19236.268} C_VEL
LIN {X 0,Y 257.204,Z 450.38,A -85,B 0,C 180,E1 -19239.193,E2 -19239.193} C_VEL
LIN {X 0,Y 253.193,Z 453.256,A -85,B 0,C 180,E1 -19242.222,E2 -19242.222} C_VEL
LIN {X 0,Y 249.805,Z 454.941,A -85,B 0,C 180,E1 -19245.333,E2 -19245.333} C_VEL
LIN {X 0,Y 247.074,Z 455.441,A -85,B 0,C 180,E1 -19248.515,E2 -19248.515} C_VEL
LIN {X 0,Y 244.863,Z 454.758,A -85,B 0,C 180,E1 -19251.749,E2 -19251.749} C_VEL
LIN {X 0,Y 243.44,Z 452.806,A -85,B 0,C 180,E1 -19255.032,E2 -19255.032} C_VEL
LIN {X 0,Y 242.606,Z 449.594,A -85,B 0,C 180,E1 -19258.34,E2 -19258.34} C_VEL
LIN {X 0,Y 242.276,Z 445.066,A -85,B 0,C 180,E1 -19261.663,E2 -19261.663} C_VEL
LIN {X 0,Y 242.047,Z 439.122,A -85,B 0,C 180,E1 -19264.998,E2 -19264.998} C_VEL
LIN {X 0,Y 242.656,Z 432.585,A -85,B 0,C 180,E1 -19267.908,E2 -19267.908} C_VEL
LIN {X 0,Y 243.326,Z 425.372,A -85,B 0,C 180,E1 -19270.574,E2 -19270.574} C_VEL
LIN {X 0,Y 244.299,Z 416.562,A -85,B 0,C 180,E1 -19273.306,E2 -19273.306} C_VEL
LIN {X 0,Y 245.51,Z 407.031,A -85,B 0,C 180,E1 -19275.781,E2 -19275.781} C_VEL
LIN {X 0,Y 246.928,Z 395.748,A -85,B 0,C 180,E1 -19278.245,E2 -19278.245} C_VEL
LIN {X 0,Y 248.668,Z 383.396,A -85,B 0,C 180,E1 -19280.473,E2 -19280.473} C_VEL
LIN {X 0,Y 249.94,Z 372.798,A -85,B 0,C 180,E1 -19282.091,E2 -19282.091} C_VEL
LIN {X 0,Y 247.08,Z 361.684,A -85,B 0,C 180,E1 -19283.762,E2 -19283.762} C_VEL
LIN {X 0,Y 243.022,Z 346.534,A -85,B 0,C 180,E1 -19285.709,E2 -19285.709} C_VEL
LIN {X 0,Y 242.209,Z 343.575,A -85,B 0,C 180,E1 -19286.113,E2 -19286.113} C_VEL
LIN {X 0,Y 242.103,Z 343.018,A -85,B 0,C 180,E1 -19286.357,E2 -19286.357} C_VEL
LIN {X 0,Y 242.037,Z 342.96,A -85,B 0,C 180,E1 -19289.58,E2 -19289.58} C_VEL
LIN {X 0,Y 241.987,Z 342.965,A -85,B 0,C 180,E1 -19293.492,E2 -19293.492} C_VEL
LIN {X 0,Y 241.995,Z 342.962,A -85,B 0,C 180,E1 -19297.582,E2 -19297.582} C_VEL
LIN {X 0,Y 241.943,Z 342.971,A -85,B 0,C 180,E1 -19301.922,E2 -19301.922} C_VEL
LIN {X 0,Y 241.949,Z 342.972,A -85,B 0,C 180,E1 -19306.569,E2 -19306.569} C_VEL
LIN {X 0,Y 241.988,Z 342.969,A -85,B 0,C 180,E1 -19310.285,E2 -19310.285} C_VEL
LIN {X 0,Y 242.043,Z 342.96,A -85,B 0,C 180,E1 -19314.497,E2 -19314.497} C_VEL
LIN {X 0,Y 241.981,Z 342.968,A -85,B 0,C 180,E1 -19318.479,E2 -19318.479} C_VEL
LIN {X 0,Y 242.007,Z 342.964,A -85,B 0,C 180,E1 -19322.311,E2 -19322.311} C_VEL
LIN {X 0,Y 242.047,Z 342.961,A -85,B 0,C 180,E1 -19326.013,E2 -19326.013} C_VEL
LIN {X 0,Y 242.042,Z 342.958,A -85,B 0,C 180,E1 -19329.607,E2 -19329.607} C_VEL
LIN {X 0,Y 242.169,Z 342.942,A -85,B 0,C 180,E1 -19333.277,E2 -19333.277} C_VEL
LIN {X 0,Y 242.192,Z 342.939,A -85,B 0,C 180,E1 -19338.279,E2 -19338.279} C_VEL
LIN {X 0,Y 242.44,Z 342.91,A -85,B 0,C 180,E1 -19341.665,E2 -19341.665} C_VEL
LIN {X 0,Y 242.265,Z 342.93,A -85,B 0,C 180,E1 -19345.006,E2 -19345.006} C_VEL
LIN {X 0,Y 242.641,Z 342.882,A -85,B 0,C 180,E1 -19348.339,E2 -19348.339} C_VEL
LIN {X 0,Y 242.64,Z 342.887,A -85,B 0,C 180,E1 -19351.658,E2 -19351.658} C_VEL
LIN {X 0,Y 242.438,Z 342.906,A -85,B 0,C 180,E1 -19356.657,E2 -19356.657} C_VEL
LIN {X 0,Y 242.348,Z 342.921,A -85,B 0,C 180,E1 -19360.019,E2 -19360.019} C_VEL
LIN {X 0,Y 242.169,Z 342.941,A -85,B 0,C 180,E1 -19365.139,E2 -19365.139} C_VEL
LIN {X 0,Y 242.075,Z 342.954,A -85,B 0,C 180,E1 -19368.622,E2 -19368.622} C_VEL
LIN {X 0,Y 242.014,Z 342.96,A -85,B 0,C 180,E1 -19372.178,E2 -19372.178} C_VEL
LIN {X 0,Y 242.067,Z 342.956,A -85,B 0,C 180,E1 -19375.836,E2 -19375.836} C_VEL
LIN {X 0,Y 242.007,Z 342.964,A -85,B 0,C 180,E1 -19379.581,E2 -19379.581} C_VEL
LIN {X 0,Y 241.979,Z 342.968,A -85,B 0,C 180,E1 -19383.491,E2 -19383.491} C_VEL
LIN {X 0,Y 241.984,Z 342.966,A -85,B 0,C 180,E1 -19387.581,E2 -19387.581} C_VEL
LIN {X 0,Y 241.936,Z 342.97,A -85,B 0,C 180,E1 -19391.92,E2 -19391.92} C_VEL
LIN {X 0,Y 241.934,Z 342.973,A -85,B 0,C 180,E1 -19396.569,E2 -19396.569} C_VEL
LIN {X 0,Y 241.952,Z 342.968,A -85,B 0,C 180,E1 -19400.279,E2 -19400.279} C_VEL
LIN {X 0,Y 241.977,Z 342.968,A -85,B 0,C 180,E1 -19404.487,E2 -19404.487} C_VEL
LIN {X 0,Y 241.97,Z 342.966,A -85,B 0,C 180,E1 -19408.479,E2 -19408.479} C_VEL
LIN {X 0,Y 242.004,Z 342.964,A -85,B 0,C 180,E1 -19412.312,E2 -19412.312} C_VEL
LIN {X 0,Y 242.052,Z 342.955,A -85,B 0,C 180,E1 -19416.015,E2 -19416.015} C_VEL
LIN {X 0,Y 242.032,Z 342.959,A -85,B 0,C 180,E1 -19419.607,E2 -19419.607} C_VEL
LIN {X 0,Y 242.157,Z 342.943,A -85,B 0,C 180,E1 -19423.277,E2 -19423.277} C_VEL
LIN {X 0,Y 242.18,Z 342.943,A -85,B 0,C 180,E1 -19428.279,E2 -19428.279} C_VEL
LIN {X 0,Y 242.429,Z 342.909,A -85,B 0,C 180,E1 -19431.665,E2 -19431.665} C_VEL
LIN {X 0,Y 242.256,Z 342.932,A -85,B 0,C 180,E1 -19435.007,E2 -19435.007} C_VEL
LIN {X 0,Y 242.63,Z 342.889,A -85,B 0,C 180,E1 -19438.34,E2 -19438.34} C_VEL
LIN {X 0,Y 242.63,Z 342.883,A -85,B 0,C 180,E1 -19441.659,E2 -19441.659} C_VEL
LIN {X 0,Y 242.427,Z 342.912,A -85,B 0,C 180,E1 -19446.659,E2 -19446.659} C_VEL
LIN {X 0,Y 242.338,Z 342.922,A -85,B 0,C 180,E1 -19450.02,E2 -19450.02} C_VEL
LIN {X 0,Y 242.16,Z 342.943,A -85,B 0,C 180,E1 -19455.141,E2 -19455.141} C_VEL
LIN {X 0,Y 242.066,Z 342.953,A -85,B 0,C 180,E1 -19458.624,E2 -19458.624} C_VEL
LIN {X 0,Y 242.006,Z 342.966,A -85,B 0,C 180,E1 -19462.18,E2 -19462.18} C_VEL
LIN {X 0,Y 242.06,Z 342.959,A -85,B 0,C 180,E1 -19465.839,E2 -19465.839} C_VEL
LIN {X 0,Y 242.022,Z 342.961,A -85,B 0,C 180,E1 -19469.581,E2 -19469.581} C_VEL
LIN {X 0,Y 242.076,Z 343.089,A -85,B 0,C 180,E1 -19474.796,E2 -19474.796} C_VEL
LIN {X 0,Y 243.467,Z 350.519,A -85,B 0,C 180,E1 -19479.424,E2 -19479.424} C_VEL
LIN {X 0,Y 245.126,Z 358.65,A -85,B 0,C 180,E1 -19484.214,E2 -19484.214} C_VEL
LIN {X 0,Y 246.645,Z 366.224,A -85,B 0,C 180,E1 -19488.471,E2 -19488.471} C_VEL
LIN {X 0,Y 245.794,Z 371.021,A -85,B 0,C 180,E1 -19491.022,E2 -19491.022} C_VEL
LIN {X 0,Y 244.739,Z 376.058,A -85,B 0,C 180,E1 -19493.672,E2 -19493.672} C_VEL
LIN {X 0,Y 243.749,Z 377.647,A -85,B 0,C 180,E1 -19494.494,E2 -19494.494} C_VEL
LIN {X 0,Y 240.43,Z 380.111,A -85,B 0,C 180,E1 -19495.755,E2 -19495.755} C_VEL
LIN {X 0,Y 237.141,Z 382.542,A -85,B 0,C 180,E1 -19497.048,E2 -19497.048} C_VEL
LIN {X 0,Y 236.226,Z 384.127,A -85,B 0,C 180,E1 -19497.907,E2 -19497.907} C_VEL
LIN {X 0,Y 235.624,Z 388.197,A -85,B 0,C 180,E1 -19499.987,E2 -19499.987} C_VEL
LIN {X 0,Y 236.54,Z 408.605,A -85,B 0,C 180,E1 -19501.618,E2 -19501.618} C_VEL
LIN {X 0,Y 237.484,Z 423.87,A -85,B 0,C 180,E1 -19503.2,E2 -19503.2} C_VEL
LIN {X 0,Y 238.361,Z 438.958,A -85,B 0,C 180,E1 -19505.157,E2 -19505.157} C_VEL
LIN {X 0,Y 239.264,Z 452.749,A -85,B 0,C 180,E1 -19507.325,E2 -19507.325} C_VEL
LIN {X 0,Y 239.19,Z 456.508,A -85,B 0,C 180,E1 -19508.001,E2 -19508.001} C_VEL
LIN {X 0,Y 237.733,Z 467.096,A -85,B 0,C 180,E1 -19510.127,E2 -19510.127} C_VEL
LIN {X 0,Y 236.258,Z 477.698,A -85,B 0,C 180,E1 -19512.696,E2 -19512.696} C_VEL
LIN {X 0,Y 235.418,Z 486.559,A -85,B 0,C 180,E1 -19515.302,E2 -19515.302} C_VEL
LIN {X 0,Y 234.923,Z 494.994,A -85,B 0,C 180,E1 -19518.352,E2 -19518.352} C_VEL
LIN {X 0,Y 235.051,Z 501.787,A -85,B 0,C 180,E1 -19521.404,E2 -19521.404} C_VEL
LIN {X 0,Y 235.354,Z 506.377,A -85,B 0,C 180,E1 -19524.002,E2 -19524.002} C_VEL
LIN {X 0,Y 235.752,Z 509.873,A -85,B 0,C 180,E1 -19526.583,E2 -19526.583} C_VEL
LIN {X 0,Y 235.955,Z 511.635,A -85,B 0,C 180,E1 -19528.295,E2 -19528.295} C_VEL
LIN {X 0,Y 236.186,Z 512.978,A -85,B 0,C 180,E1 -19530.002,E2 -19530.002} C_VEL
LIN {X 0,Y 235.636,Z 513.734,A -85,B 0,C 180,E1 -19531.711,E2 -19531.711} C_VEL
LIN {X 0,Y 234.58,Z 514.161,A -85,B 0,C 180,E1 -19535.158,E2 -19535.158} C_VEL
LIN {X 0,Y 234.012,Z 513.612,A -85,B 0,C 180,E1 -19537.661,E2 -19537.661} C_VEL
LIN {X 0,Y 233.692,Z 512.3,A -85,B 0,C 180,E1 -19540.397,E2 -19540.397} C_VEL
LIN {X 0,Y 234.075,Z 509.556,A -85,B 0,C 180,E1 -19543.9,E2 -19543.9} C_VEL
LIN {X 0,Y 235.977,Z 504.564,A -85,B 0,C 180,E1 -19548.225,E2 -19548.225} C_VEL
LIN {X 0,Y 238.636,Z 499.253,A -85,B 0,C 180,E1 -19551.602,E2 -19551.602} C_VEL
LIN {X 0,Y 242.463,Z 492.792,A -85,B 0,C 180,E1 -19554.855,E2 -19554.855} C_VEL
LIN {X 0,Y 247.693,Z 484.343,A -85,B 0,C 180,E1 -19558.268,E2 -19558.268} C_VEL
LIN {X 0,Y 253.929,Z 474.976,A -85,B 0,C 180,E1 -19561.263,E2 -19561.263} C_VEL
LIN {X 0,Y 259.801,Z 464.722,A -85,B 0,C 180,E1 -19564.148,E2 -19564.148} C_VEL
LIN {X 0,Y 264.144,Z 456.674,A -85,B 0,C 180,E1 -19566.184,E2 -19566.184} C_VEL
LIN {X 0,Y 268.007,Z 448.277,A -85,B 0,C 180,E1 -19568.39,E2 -19568.39} C_VEL
LIN {X 0,Y 271.579,Z 439.722,A -85,B 0,C 180,E1 -19570.78,E2 -19570.78} C_VEL
LIN {X 0,Y 275.112,Z 430.898,A -85,B 0,C 180,E1 -19573.611,E2 -19573.611} C_VEL
LIN {X 0,Y 278.192,Z 424.198,A -85,B 0,C 180,E1 -19576.06,E2 -19576.06} C_VEL
LIN {X 0,Y 279.101,Z 422.169,A -85,B 0,C 180,E1 -19577.166,E2 -19577.166} C_VEL
LIN {X 0,Y 279.5,Z 420.728,A -85,B 0,C 180,E1 -19579.174,E2 -19579.174} C_VEL
LIN {X 0,Y 280.123,Z 420.006,A -85,B 0,C 180,E1 -19581.155,E2 -19581.155} C_VEL
LIN {X 0,Y 280.869,Z 419.986,A -85,B 0,C 180,E1 -19583.2,E2 -19583.2} C_VEL
LIN {X 0,Y 281.301,Z 420.878,A -85,B 0,C 180,E1 -19584.927,E2 -19584.927} C_VEL
LIN {X 0,Y 280.457,Z 422.402,A -85,B 0,C 180,E1 -19585.679,E2 -19585.679} C_VEL
LIN {X 0,Y 273.077,Z 431.573,A -85,B 0,C 180,E1 -19588.156,E2 -19588.156} C_VEL
LIN {X 0,Y 266.248,Z 439.073,A -85,B 0,C 180,E1 -19590.769,E2 -19590.769} C_VEL
LIN {X 0,Y 259.825,Z 445.342,A -85,B 0,C 180,E1 -19593.6,E2 -19593.6} C_VEL
LIN {X 0,Y 254.585,Z 449.872,A -85,B 0,C 180,E1 -19596.405,E2 -19596.405} C_VEL
LIN {X 0,Y 250.925,Z 452.602,A -85,B 0,C 180,E1 -19598.648,E2 -19598.648} C_VEL
LIN {X 0,Y 246.695,Z 455.164,A -85,B 0,C 180,E1 -19601.738,E2 -19601.738} C_VEL
LIN {X 0,Y 243.151,Z 456.559,A -85,B 0,C 180,E1 -19604.922,E2 -19604.922} C_VEL
LIN {X 0,Y 240.263,Z 456.799,A -85,B 0,C 180,E1 -19608.185,E2 -19608.185} C_VEL
LIN {X 0,Y 237.933,Z 455.869,A -85,B 0,C 180,E1 -19611.507,E2 -19611.507} C_VEL
LIN {X 0,Y 236.447,Z 453.681,A -85,B 0,C 180,E1 -19614.885,E2 -19614.885} C_VEL
LIN {X 0,Y 235.539,Z 450.246,A -85,B 0,C 180,E1 -19618.291,E2 -19618.291} C_VEL
LIN {X 0,Y 235.186,Z 445.495,A -85,B 0,C 180,E1 -19621.713,E2 -19621.713} C_VEL
LIN {X 0,Y 235,Z 439.325,A -85,B 0,C 180,E1 -19625.148,E2 -19625.148} C_VEL
LIN {X 0,Y 235.655,Z 432.103,A -85,B 0,C 180,E1 -19628.322,E2 -19628.322} C_VEL
LIN {X 0,Y 236.469,Z 424.039,A -85,B 0,C 180,E1 -19631.247,E2 -19631.247} C_VEL
LIN {X 0,Y 237.557,Z 414.469,A -85,B 0,C 180,E1 -19634.128,E2 -19634.128} C_VEL
LIN {X 0,Y 238.834,Z 404.373,A -85,B 0,C 180,E1 -19636.673,E2 -19636.673} C_VEL
LIN {X 0,Y 240.436,Z 392.42,A -85,B 0,C 180,E1 -19639.199,E2 -19639.199} C_VEL
LIN {X 0,Y 242.259,Z 379.02,A -85,B 0,C 180,E1 -19641.512,E2 -19641.512} C_VEL
LIN {X 0,Y 242.886,Z 373.678,A -85,B 0,C 180,E1 -19642.32,E2 -19642.32} C_VEL
LIN {X 0,Y 239.606,Z 361.094,A -85,B 0,C 180,E1 -19644.246,E2 -19644.246} C_VEL
LIN {X 0,Y 235.783,Z 346.792,A -85,B 0,C 180,E1 -19646.122,E2 -19646.122} C_VEL
LIN {X 0,Y 235.114,Z 344.252,A -85,B 0,C 180,E1 -19646.516,E2 -19646.516} C_VEL
LIN {X 0,Y 235.028,Z 343.848,A -85,B 0,C 180,E1 -19646.891,E2 -19646.891} C_VEL
LIN {X 0,Y 234.938,Z 343.847,A -85,B 0,C 180,E1 -19650.568,E2 -19650.568} C_VEL
LIN {X 0,Y 234.936,Z 343.847,A -85,B 0,C 180,E1 -19654.638,E2 -19654.638} C_VEL
LIN {X 0,Y 234.948,Z 343.843,A -85,B 0,C 180,E1 -19658.944,E2 -19658.944} C_VEL
LIN {X 0,Y 234.894,Z 343.847,A -85,B 0,C 180,E1 -19663.485,E2 -19663.485} C_VEL
LIN {X 0,Y 234.927,Z 343.847,A -85,B 0,C 180,E1 -19666.521,E2 -19666.521} C_VEL
LIN {X 0,Y 234.961,Z 343.84,A -85,B 0,C 180,E1 -19671.085,E2 -19671.085} C_VEL
LIN {X 0,Y 234.967,Z 343.838,A -85,B 0,C 180,E1 -19675.367,E2 -19675.367} C_VEL
LIN {X 0,Y 234.929,Z 343.844,A -85,B 0,C 180,E1 -19679.43,E2 -19679.43} C_VEL
LIN {X 0,Y 234.999,Z 343.835,A -85,B 0,C 180,E1 -19683.793,E2 -19683.793} C_VEL
LIN {X 0,Y 235.004,Z 343.834,A -85,B 0,C 180,E1 -19688.968,E2 -19688.968} C_VEL
LIN {X 0,Y 235.102,Z 343.822,A -85,B 0,C 180,E1 -19693.058,E2 -19693.058} C_VEL
LIN {X 0,Y 235.152,Z 343.818,A -85,B 0,C 180,E1 -19697.923,E2 -19697.923} C_VEL
LIN {X 0,Y 235.396,Z 343.786,A -85,B 0,C 180,E1 -19701.413,E2 -19701.413} C_VEL
LIN {X 0,Y 235.411,Z 343.784,A -85,B 0,C 180,E1 -19703.14,E2 -19703.14} C_VEL
LIN {X 0,Y 235.6,Z 343.759,A -85,B 0,C 180,E1 -19708.289,E2 -19708.289} C_VEL
LIN {X 0,Y 235.6,Z 343.764,A -85,B 0,C 180,E1 -19711.708,E2 -19711.708} C_VEL
LIN {X 0,Y 235.41,Z 343.782,A -85,B 0,C 180,E1 -19716.857,E2 -19716.857} C_VEL
LIN {X 0,Y 235.256,Z 343.804,A -85,B 0,C 180,E1 -19720.324,E2 -19720.324} C_VEL
LIN {X 0,Y 235.116,Z 343.822,A -85,B 0,C 180,E1 -19725.604,E2 -19725.604} C_VEL
LIN {X 0,Y 235.011,Z 343.836,A -85,B 0,C 180,E1 -19729.204,E2 -19729.204} C_VEL
LIN {X 0,Y 234.962,Z 343.839,A -85,B 0,C 180,E1 -19732.881,E2 -19732.881} C_VEL
LIN {X 0,Y 234.968,Z 343.839,A -85,B 0,C 180,E1 -19736.656,E2 -19736.656} C_VEL
LIN {X 0,Y 234.922,Z 343.844,A -85,B 0,C 180,E1 -19740.567,E2 -19740.567} C_VEL
LIN {X 0,Y 234.925,Z 343.845,A -85,B 0,C 180,E1 -19744.637,E2 -19744.637} C_VEL
LIN {X 0,Y 234.94,Z 343.845,A -85,B 0,C 180,E1 -19748.943,E2 -19748.943} C_VEL
LIN {X 0,Y 234.887,Z 343.851,A -85,B 0,C 180,E1 -19753.483,E2 -19753.483} C_VEL
LIN {X 0,Y 234.886,Z 343.85,A -85,B 0,C 180,E1 -19756.513,E2 -19756.513} C_VEL
LIN {X 0,Y 234.915,Z 343.849,A -85,B 0,C 180,E1 -19761.077,E2 -19761.077} C_VEL
LIN {X 0,Y 234.922,Z 343.845,A -85,B 0,C 180,E1 -19765.36,E2 -19765.36} C_VEL
LIN {X 0,Y 234.927,Z 343.844,A -85,B 0,C 180,E1 -19769.431,E2 -19769.431} C_VEL
LIN {X 0,Y 234.989,Z 343.836,A -85,B 0,C 180,E1 -19773.792,E2 -19773.792} C_VEL
LIN {X 0,Y 235.006,Z 343.837,A -85,B 0,C 180,E1 -19778.969,E2 -19778.969} C_VEL
LIN {X 0,Y 235.09,Z 343.824,A -85,B 0,C 180,E1 -19783.058,E2 -19783.058} C_VEL
LIN {X 0,Y 235.14,Z 343.818,A -85,B 0,C 180,E1 -19787.923,E2 -19787.923} C_VEL
LIN {X 0,Y 235.384,Z 343.786,A -85,B 0,C 180,E1 -19791.414,E2 -19791.414} C_VEL
LIN {X 0,Y 235.399,Z 343.783,A -85,B 0,C 180,E1 -19793.141,E2 -19793.141} C_VEL
LIN {X 0,Y 235.59,Z 343.765,A -85,B 0,C 180,E1 -19798.29,E2 -19798.29} C_VEL
LIN {X 0,Y 235.59,Z 343.76,A -85,B 0,C 180,E1 -19801.709,E2 -19801.709} C_VEL
LIN {X 0,Y 235.399,Z 343.786,A -85,B 0,C 180,E1 -19806.858,E2 -19806.858} C_VEL
LIN {X 0,Y 235.246,Z 343.805,A -85,B 0,C 180,E1 -19810.326,E2 -19810.326} C_VEL
LIN {X 0,Y 235.107,Z 343.823,A -85,B 0,C 180,E1 -19815.606,E2 -19815.606} C_VEL
LIN {X 0,Y 235.002,Z 343.832,A -85,B 0,C 180,E1 -19819.206,E2 -19819.206} C_VEL
LIN {X 0,Y 234.954,Z 343.841,A -85,B 0,C 180,E1 -19822.883,E2 -19822.883} C_VEL
LIN {X 0,Y 234.962,Z 343.838,A -85,B 0,C 180,E1 -19826.658,E2 -19826.658} C_VEL
LIN {X 0,Y 234.925,Z 343.845,A -85,B 0,C 180,E1 -19830.568,E2 -19830.568} C_VEL
LIN {X 0,Y 235.041,Z 344.021,A -85,B 0,C 180,E1 -19834.619,E2 -19834.619} C_VEL
LIN {X 0,Y 236.439,Z 351.509,A -85,B 0,C 180,E1 -19839.394,E2 -19839.394} C_VEL
LIN {X 0,Y 237.988,Z 358.928,A -85,B 0,C 180,E1 -19843.896,E2 -19843.896} C_VEL
LIN {X 0,Y 239.487,Z 366.196,A -85,B 0,C 180,E1 -19848.119,E2 -19848.119} C_VEL
LIN {X 0,Y 239.145,Z 369.279,A -85,B 0,C 180,E1 -19849.826,E2 -19849.826} C_VEL
LIN {X 0,Y 237.597,Z 376.451,A -85,B 0,C 180,E1 -19853.732,E2 -19853.732} C_VEL
LIN {X 0,Y 236.226,Z 384.127,A -85,B 0,C 180,E1 -19857.907,E2 -19857.907} C_VEL
LIN {X 0,Y 235.723,Z 386.176,A -85,B 0,C 180,E1 -19858.682,E2 -19858.682} C_VEL
LIN {X 0,Y 234.54,Z 389.665,A -85,B 0,C 180,E1 -19859.448,E2 -19859.448} C_VEL
LIN {X 0,Y 232.467,Z 395.478,A -85,B 0,C 180,E1 -19860.216,E2 -19860.216} C_VEL
LIN {X 0,Y 230.282,Z 403.085,A -85,B 0,C 180,E1 -19860.877,E2 -19860.877} C_VEL
LIN {X 0,Y 229.581,Z 408.909,A -85,B 0,C 180,E1 -19861.375,E2 -19861.375} C_VEL
LIN {X 0,Y 229.647,Z 410.827,A -85,B 0,C 180,E1 -19861.565,E2 -19861.565} C_VEL
LIN {X 0,Y 230.502,Z 425.99,A -85,B 0,C 180,E1 -19863.276,E2 -19863.276} C_VEL
LIN {X 0,Y 231.342,Z 440.546,A -85,B 0,C 180,E1 -19865.294,E2 -19865.294} C_VEL
LIN {X 0,Y 232.249,Z 453.865,A -85,B 0,C 180,E1 -19867.542,E2 -19867.542} C_VEL
LIN {X 0,Y 231.144,Z 462.737,A -85,B 0,C 180,E1 -19869.303,E2 -19869.303} C_VEL
LIN {X 0,Y 229.737,Z 473.298,A -85,B 0,C 180,E1 -19871.805,E2 -19871.805} C_VEL
LIN {X 0,Y 228.58,Z 483.815,A -85,B 0,C 180,E1 -19874.852,E2 -19874.852} C_VEL
LIN {X 0,Y 228.031,Z 492.593,A -85,B 0,C 180,E1 -19877.994,E2 -19877.994} C_VEL
LIN {X 0,Y 228.076,Z 499.613,A -85,B 0,C 180,E1 -19881.139,E2 -19881.139} C_VEL
LIN {X 0,Y 228.386,Z 504.362,A -85,B 0,C 180,E1 -19883.819,E2 -19883.819} C_VEL
LIN {X 0,Y 228.808,Z 508.021,A -85,B 0,C 180,E1 -19886.48,E2 -19886.48} C_VEL
LIN {X 0,Y 229.039,Z 509.882,A -85,B 0,C 180,E1 -19888.243,E2 -19888.243} C_VEL
LIN {X 0,Y 229.256,Z 511.313,A -85,B 0,C 180,E1 -19890.002,E2 -19890.002} C_VEL
LIN {X 0,Y 228.675,Z 512.155,A -85,B 0,C 180,E1 -19891.763,E2 -19891.763} C_VEL
LIN {X 0,Y 227.558,Z 512.741,A -85,B 0,C 180,E1 -19895.318,E2 -19895.318} C_VEL
LIN {X 0,Y 226.796,Z 512.003,A -85,B 0,C 180,E1 -19898.915,E2 -19898.915} C_VEL
LIN {X 0,Y 226.764,Z 510.063,A -85,B 0,C 180,E1 -19902.531,E2 -19902.531} C_VEL
LIN {X 0,Y 227.741,Z 507.002,A -85,B 0,C 180,E1 -19906.127,E2 -19906.127} C_VEL
LIN {X 0,Y 229.761,Z 502.83,A -85,B 0,C 180,E1 -19909.664,E2 -19909.664} C_VEL
LIN {X 0,Y 232.845,Z 497.541,A -85,B 0,C 180,E1 -19913.104,E2 -19913.104} C_VEL
LIN {X 0,Y 238.406,Z 489.363,A -85,B 0,C 180,E1 -19917.19,E2 -19917.19} C_VEL
LIN {X 0,Y 243.136,Z 482.558,A -85,B 0,C 180,E1 -19919.91,E2 -19919.91} C_VEL
LIN {X 0,Y 247.945,Z 475.939,A -85,B 0,C 180,E1 -19922.106,E2 -19922.106} C_VEL
LIN {X 0,Y 254.924,Z 464.945,A -85,B 0,C 180,E1 -19925.378,E2 -19925.378} C_VEL
LIN {X 0,Y 259.481,Z 457.267,A -85,B 0,C 180,E1 -19927.461,E2 -19927.461} C_VEL
LIN {X 0,Y 264.291,Z 447.773,A -85,B 0,C 180,E1 -19930.156,E2 -19930.156} C_VEL
LIN {X 0,Y 267.788,Z 440.375,A -85,B 0,C 180,E1 -19932.446,E2 -19932.446} C_VEL
LIN {X 0,Y 271.968,Z 431.841,A -85,B 0,C 180,E1 -19935.485,E2 -19935.485} C_VEL
LIN {X 0,Y 274.021,Z 428.136,A -85,B 0,C 180,E1 -19937.032,E2 -19937.032} C_VEL
LIN {X 0,Y 274.55,Z 426.744,A -85,B 0,C 180,E1 -19938.275,E2 -19938.275} C_VEL
LIN {X 0,Y 275.068,Z 425.599,A -85,B 0,C 180,E1 -19940.302,E2 -19940.302} C_VEL
LIN {X 0,Y 275.654,Z 425.204,A -85,B 0,C 180,E1 -19942.274,E2 -19942.274} C_VEL
LIN {X 0,Y 276.199,Z 425.734,A -85,B 0,C 180,E1 -19944.515,E2 -19944.515} C_VEL
LIN {X 0,Y 275.449,Z 426.764,A -85,B 0,C 180,E1 -19944.964,E2 -19944.964} C_VEL
LIN {X 0,Y 267.764,Z 435.303,A -85,B 0,C 180,E1 -19947.448,E2 -19947.448} C_VEL
LIN {X 0,Y 260.667,Z 442.352,A -85,B 0,C 180,E1 -19950.08,E2 -19950.08} C_VEL
LIN {X 0,Y 254.175,Z 448.038,A -85,B 0,C 180,E1 -19952.856,E2 -19952.856} C_VEL
LIN {X 0,Y 249.857,Z 451.368,A -85,B 0,C 180,E1 -19955.044,E2 -19955.044} C_VEL
LIN {X 0,Y 244.675,Z 454.807,A -85,B 0,C 180,E1 -19958.074,E2 -19958.074} C_VEL
LIN {X 0,Y 240.23,Z 457.066,A -85,B 0,C 180,E1 -19961.228,E2 -19961.228} C_VEL
LIN {X 0,Y 236.498,Z 458.183,A -85,B 0,C 180,E1 -19964.488,E2 -19964.488} C_VEL
LIN {X 0,Y 233.455,Z 458.158,A -85,B 0,C 180,E1 -19967.835,E2 -19967.835} C_VEL
LIN {X 0,Y 231.006,Z 456.97,A -85,B 0,C 180,E1 -19971.251,E2 -19971.251} C_VEL
LIN {X 0,Y 229.43,Z 454.539,A -85,B 0,C 180,E1 -19974.728,E2 -19974.728} C_VEL
LIN {X 0,Y 228.47,Z 450.869,A -85,B 0,C 180,E1 -19978.238,E2 -19978.238} C_VEL
LIN {X 0,Y 228.094,Z 445.866,A -85,B 0,C 180,E1 -19981.766,E2 -19981.766} C_VEL
LIN {X 0,Y 227.939,Z 439.393,A -85,B 0,C 180,E1 -19985.308,E2 -19985.308} C_VEL
LIN {X 0,Y 228.59,Z 432.29,A -85,B 0,C 180,E1 -19988.436,E2 -19988.436} C_VEL
LIN {X 0,Y 229.409,Z 424.257,A -85,B 0,C 180,E1 -19991.378,E2 -19991.378} C_VEL
LIN {X 0,Y 230.626,Z 413.771,A -85,B 0,C 180,E1 -19994.561,E2 -19994.561} C_VEL
LIN {X 0,Y 231.943,Z 403.39,A -85,B 0,C 180,E1 -19997.184,E2 -19997.184} C_VEL
LIN {X 0,Y 233.693,Z 390.961,A -85,B 0,C 180,E1 -19999.776,E2 -19999.776} C_VEL
LIN {X 0,Y 235.383,Z 378.342,A -85,B 0,C 180,E1 -20001.963,E2 -20001.963} C_VEL
LIN {X 0,Y 235.768,Z 374.018,A -85,B 0,C 180,E1 -20002.633,E2 -20002.633} C_VEL
LIN {X 0,Y 232.146,Z 360.531,A -85,B 0,C 180,E1 -20004.736,E2 -20004.736} C_VEL
LIN {X 0,Y 228.082,Z 345.301,A -85,B 0,C 180,E1 -20006.812,E2 -20006.812} C_VEL
LIN {X 0,Y 227.956,Z 344.748,A -85,B 0,C 180,E1 -20007.143,E2 -20007.143} C_VEL
LIN {X 0,Y 227.877,Z 344.724,A -85,B 0,C 180,E1 -20011.622,E2 -20011.622} C_VEL
LIN {X 0,Y 227.887,Z 344.721,A -85,B 0,C 180,E1 -20015.871,E2 -20015.871} C_VEL
LIN {X 0,Y 227.832,Z 344.731,A -85,B 0,C 180,E1 -20020.376,E2 -20020.376} C_VEL
LIN {X 0,Y 227.842,Z 344.724,A -85,B 0,C 180,E1 -20025.192,E2 -20025.192} C_VEL
LIN {X 0,Y 227.846,Z 344.727,A -85,B 0,C 180,E1 -20029.626,E2 -20029.626} C_VEL
LIN {X 0,Y 227.907,Z 344.719,A -85,B 0,C 180,E1 -20034.131,E2 -20034.131} C_VEL
LIN {X 0,Y 227.875,Z 344.726,A -85,B 0,C 180,E1 -20038.377,E2 -20038.377} C_VEL
LIN {X 0,Y 227.885,Z 344.722,A -85,B 0,C 180,E1 -20042.443,E2 -20042.443} C_VEL
LIN {X 0,Y 227.912,Z 344.72,A -85,B 0,C 180,E1 -20046.366,E2 -20046.366} C_VEL
LIN {X 0,Y 227.943,Z 344.714,A -85,B 0,C 180,E1 -20050.173,E2 -20050.173} C_VEL
LIN {X 0,Y 228.063,Z 344.702,A -85,B 0,C 180,E1 -20053.897,E2 -20053.897} C_VEL
LIN {X 0,Y 228.177,Z 344.683,A -85,B 0,C 180,E1 -20059.349,E2 -20059.349} C_VEL
LIN {X 0,Y 228.363,Z 344.662,A -85,B 0,C 180,E1 -20062.927,E2 -20062.927} C_VEL
LIN {X 0,Y 228.559,Z 344.637,A -85,B 0,C 180,E1 -20068.236,E2 -20068.236} C_VEL
LIN {X 0,Y 228.559,Z 344.642,A -85,B 0,C 180,E1 -20071.76,E2 -20071.76} C_VEL
LIN {X 0,Y 228.362,Z 344.66,A -85,B 0,C 180,E1 -20077.07,E2 -20077.07} C_VEL
LIN {X 0,Y 228.175,Z 344.686,A -85,B 0,C 180,E1 -20080.648,E2 -20080.648} C_VEL
LIN {X 0,Y 228.06,Z 344.699,A -85,B 0,C 180,E1 -20086.1,E2 -20086.1} C_VEL
LIN {X 0,Y 227.944,Z 344.716,A -85,B 0,C 180,E1 -20089.823,E2 -20089.823} C_VEL
LIN {X 0,Y 227.915,Z 344.718,A -85,B 0,C 180,E1 -20093.631,E2 -20093.631} C_VEL
LIN {X 0,Y 227.879,Z 344.725,A -85,B 0,C 180,E1 -20097.554,E2 -20097.554} C_VEL
LIN {X 0,Y 227.866,Z 344.723,A -85,B 0,C 180,E1 -20101.621,E2 -20101.621} C_VEL
LIN {X 0,Y 227.878,Z 344.723,A -85,B 0,C 180,E1 -20105.87,E2 -20105.87} C_VEL
LIN {X 0,Y 227.824,Z 344.727,A -85,B 0,C 180,E1 -20110.375,E2 -20110.375} C_VEL
LIN {X 0,Y 227.832,Z 344.731,A -85,B 0,C 180,E1 -20115.19,E2 -20115.19} C_VEL
LIN {X 0,Y 227.823,Z 344.728,A -85,B 0,C 180,E1 -20119.622,E2 -20119.622} C_VEL
LIN {X 0,Y 227.876,Z 344.723,A -85,B 0,C 180,E1 -20124.127,E2 -20124.127} C_VEL
LIN {X 0,Y 227.866,Z 344.722,A -85,B 0,C 180,E1 -20128.376,E2 -20128.376} C_VEL
LIN {X 0,Y 227.881,Z 344.724,A -85,B 0,C 180,E1 -20132.444,E2 -20132.444} C_VEL
LIN {X 0,Y 227.909,Z 344.718,A -85,B 0,C 180,E1 -20136.366,E2 -20136.366} C_VEL
LIN {X 0,Y 227.937,Z 344.716,A -85,B 0,C 180,E1 -20140.173,E2 -20140.173} C_VEL
LIN {X 0,Y 228.051,Z 344.699,A -85,B 0,C 180,E1 -20143.897,E2 -20143.897} C_VEL
LIN {X 0,Y 228.165,Z 344.687,A -85,B 0,C 180,E1 -20149.349,E2 -20149.349} C_VEL
LIN {X 0,Y 228.352,Z 344.661,A -85,B 0,C 180,E1 -20152.928,E2 -20152.928} C_VEL
LIN {X 0,Y 228.549,Z 344.642,A -85,B 0,C 180,E1 -20158.237,E2 -20158.237} C_VEL
LIN {X 0,Y 228.549,Z 344.637,A -85,B 0,C 180,E1 -20161.762,E2 -20161.762} C_VEL
